FUNCTION_BLOCK "TYPIC_C106_IF_TFO"   // FB80, FBD
TITLE = TYPIC_C106_IF_TFO: Transformator
{ S7_Optimized_Access := 'TRUE' }
AUTHOR : OCOTECH
FAMILY : Typical
NAME : C106.704
// Logisch Object Besturing: C106.704
// 
// De interne functie Transformator verzorgt de bewaking van een transformator.
// stored: MemoryReserve 10, SetENOAutomatically false
   VAR_INPUT
      EXT_AUT { ExternalAccessible := 'False'; ExternalVisible := 'False'; ExternalWritable := 'False'} : Bool;   // Externe (hoofd) beveiliging (1 = OK)
      EXT_HW { ExternalAccessible := 'False'; ExternalVisible := 'False'; ExternalWritable := 'False'} : Bool;   // Sturings hardware (PLC) bewaking (1 = OK)
      IN_STO_NOK { ExternalAccessible := 'False'; ExternalVisible := 'False'; ExternalWritable := 'False'} : Bool;   // Storing aanwezig die niet observeerbaar tot gevolg heeft
      IN_STO_OK { ExternalAccessible := 'False'; ExternalVisible := 'False'; ExternalWritable := 'False'} : Bool;   // Storing aanwezig die observeerbaarheid niet beinvloed
      IN_TFO_BSC1 { ExternalAccessible := 'False'; ExternalVisible := 'False'; ExternalWritable := 'False'} : Bool;   // Transformator beschikbaar
      IN_TFO_BSC2 { ExternalAccessible := 'False'; ExternalVisible := 'False'; ExternalWritable := 'False'} : Bool;   // Transformator niet beschikbaar
      IN_TFO_BSC3 { ExternalAccessible := 'False'; ExternalVisible := 'False'; ExternalWritable := 'False'} : Bool;   // Transformator beperkt beschikbaar
      IN_AUT_C106 { ExternalAccessible := 'False'; ExternalVisible := 'False'; ExternalWritable := 'False'} : Bool;   // Beveiligingen: serie geschakelde terugmelding (1 = OK)
   END_VAR
   VAR_OUTPUT
      VAR_IF_NME { ExternalAccessible := 'False'; ExternalVisible := 'False'; ExternalWritable := 'False'} : "C106_VAR_IF_NME_TYPIC";   // Struct met alle variabelen naar bovenliggende functies
   END_VAR
   VAR
      STO { ExternalWritable := 'False'} : Struct   // Storingen
         A001 : Bool;   // Beveiliging aangesproken
         A002 : Bool;   // Hoogspanningstransformator in storing
         A003 : Bool;   // Algemene storing hoogspanningstransformator
      END_STRUCT;
      VAR { ExternalWritable := 'False'} : Struct   // Variabelen
         BSC1 { ExternalAccessible := 'False'; ExternalVisible := 'False'} : Bool;   // Transformator beschikbaar
         BSC2 { ExternalAccessible := 'False'; ExternalVisible := 'False'} : Bool;   // Transformator niet beschikbaar
         BSC3 { ExternalAccessible := 'False'; ExternalVisible := 'False'} : Bool;   // Transformator beperkt beschikbaar
         EXT_AUT { ExternalAccessible := 'False'; ExternalVisible := 'False'} : Bool;   // Externe (hoofd) beveiliging aangesproken
         EXT_HW { ExternalAccessible := 'False'; ExternalVisible := 'False'} : Bool;   // Sturings hardware (PLC) in storing
      END_STRUCT;
   END_VAR
BEGIN

REGION Network 1: START
END_REGION

REGION Network 2: +++ Verwerking meetwaarden en statussen +++
   // De meetwaarde en status wordt ontvangen vanuit de interne sturing.
END_REGION

REGION Network 3: +++ Storingen +++
   // Verwerken van de storingsmeldingen (inputs).
END_REGION

REGION Network 4: Storing A001: Beveiliging aangesproken
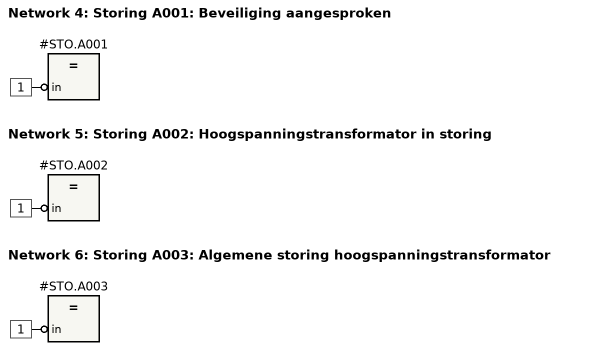
   #STO.A001 := NOT 1;
END_REGION

REGION Network 5: Storing A002: Hoogspanningstransformator in storing
   #STO.A002 := NOT 1;
END_REGION

REGION Network 6: Storing A003: Algemene storing hoogspanningstransformator
   #STO.A003 := NOT 1;
END_REGION

REGION Network 7 (SCL): EINDE
   // Variabelen van intern scada rakvlak naar outputs copieren
   #VAR_IF_NME.BSC1 := #VAR.BSC1;
   #VAR_IF_NME.BSC2 := #VAR.BSC2;
   #VAR_IF_NME.BSC3 := #VAR.BSC3;
   #VAR_IF_NME.EXT_AUT := #VAR.EXT_AUT;
   #VAR_IF_NME.EXT_HW := #VAR.EXT_HW;
END_REGION
END_FUNCTION_BLOCK

FUNCTION_BLOCK "TYPIC_C103_BF_LSK"   // FB21, FBD
TITLE = TYPIC_C103_BF_LSK: Laagspanning koker
{ S7_Optimized_Access := 'TRUE' }
AUTHOR : OCOTECH
FAMILY : Typical
NAME : C103.801
// Logisch Object Besturing: C103.801
// 
// Het doel van de BF LSK (laagspanning koker) is om de algemene opvolging te voorzien van de laagspanningsinstallatie per verkeerskoker.
// stored: MemoryReserve 10, SetENOAutomatically false
   VAR_INPUT
      STU_ALG_LCK_SIG { ExternalAccessible := 'False'; ExternalVisible := 'False'; ExternalWritable := 'False'} : USInt;   // Onderdruk alarmen
   END_VAR
   VAR_IN_OUT
      VAR_REL : Array[0..1] of Bool;   // Array met de standmeldingen van alle vermogenschakelaars
   END_VAR
   VAR
      SIG { ExternalWritable := 'False'} : Struct   // Signaleringen
         AA01 : Bool;   // Laagspanningsinstallatie niet observeerbaar
         AA02 : Bool;   // Laagspanningsinstallatie storing algemeen
         A001 : Bool;   // Laagspanningsinstallatie standmelding beveiliging uit
         AB01 : Bool;   // Laagspanningsinstallatie niet beschikbaar
         AB02 : Bool;   // Laagspanningsinstallatie beperkt beschikbaar
      END_STRUCT;
      VAR { ExternalWritable := 'False'} : Struct   // Variabelen
         BSC : USInt;   // Geeft de beschikbaarheid aan van het deelsysteem
         LSK_STS : USInt;   // De status van het deelsysteem
         VGV_SIG_VOP : Bool;   // TRUE = Signaleringen vrijgegeven voor verkeersoperator FALSE = Onderdrukt
      END_STRUCT;
   END_VAR
BEGIN

REGION Network 1: START
END_REGION

REGION Network 2: +++ Bepalen beschikbaarheidsstatus +++
   // Beschikbaarheidsstatus (beschikbaar / beperkt beschikbaar / niet beschikbaar) bepalen.
END_REGION

REGION Network 3 (SCL): Beschikbaarheidsstatus bepalen
   IF 
       //voorwaarden "Niet beschikbaar"
       TRUE
   THEN
       //Beschikbaarheidsstatus = Niet Beschikbaar
       #VAR.BSC:= "NietBeschikbaar";
   ELSIF
       //voorwaarden "Beperkt beschikbaar"
       TRUE
   THEN
       //Beschikbaarheidsstatus = Beperkt Beschikbaar
       #VAR.BSC:= "Beperkt";
   ELSE
       //Beschikbaarheidsstatus = Beschikbaar
       #VAR.BSC:= "Beschikbaar";
   END_IF;
END_REGION

REGION Network 4: +++ Signaleringen +++
   // Aanmaken signaleringen
END_REGION

REGION Network 5: Signalering AB01 : Niet Beschikbaar
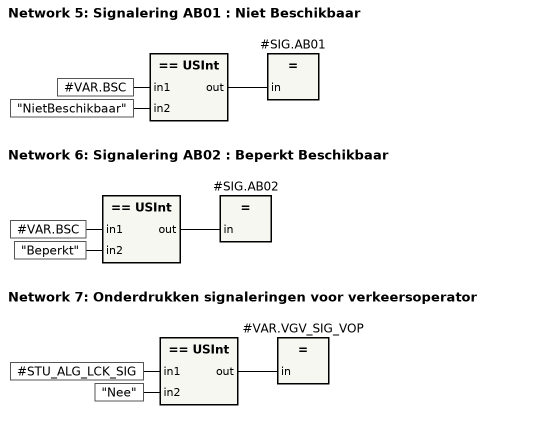
   #SIG.AB01 := #VAR.BSC = "NietBeschikbaar";
END_REGION

REGION Network 6: Signalering AB02 : Beperkt Beschikbaar
   #SIG.AB02 := #VAR.BSC = "Beperkt";
END_REGION

REGION Network 7: Onderdrukken signaleringen voor verkeersoperator
   // Via de variabele VGV_SIG_VOP wordt aan IRIS SCADA doorgegeven of signaleringen (bestemd voor de verkeersoperator) van de deze functie zichtbaar (of onderdrukt) moeten zijn.
   #VAR.VGV_SIG_VOP := #STU_ALG_LCK_SIG = "Nee";
END_REGION

REGION Network 8: +++ Doorkoppeling energieverbruik en vermogen LSK +++
   // De actuele vermogen en energiemeting wordt doorgegeven aan de coordinerende functie Energievoorziening.
END_REGION

REGION Network 9: EINDE
   // Variabelen van intern scada rakvlak naar outputs copieren
END_REGION
END_FUNCTION_BLOCK

FUNCTION_BLOCK "TYPIC_C103_IF_HVI"   // FB20, FBD
TITLE = TYPIC_C103_IF_HVI: ALSB
{ S7_Optimized_Access := 'TRUE' }
AUTHOR : OCOTECH
FAMILY : Typical
NAME : C103.701
// Logisch Object Besturing: C103.802
// 
// De interne functie laagspanningsverdeelbord verzorgt de bewaking van een laagspanningsverdeelbord.
// stored: MemoryReserve 10, SetENOAutomatically false
   VAR_INPUT
      EXT_AUT { ExternalAccessible := 'False'; ExternalVisible := 'False'; ExternalWritable := 'False'} : Bool;   // Externe (hoofd) beveiliging (1 = OK)
      EXT_HW { ExternalAccessible := 'False'; ExternalVisible := 'False'; ExternalWritable := 'False'} : Bool;   // Sturings hardware (PLC) bewaking (1 = OK)
      IN_PWR1 { ExternalAccessible := 'False'; ExternalVisible := 'False'; ExternalWritable := 'False'} : Real;   // Actief vermogen
      IN_PWR2 { ExternalAccessible := 'False'; ExternalVisible := 'False'; ExternalWritable := 'False'} : Real;   // Reactief vermogen
      IN_SPA_1 { ExternalAccessible := 'False'; ExternalVisible := 'False'; ExternalWritable := 'False'} : Real;   // Spanningsniveau lijn 1
      IN_SPA_2 { ExternalAccessible := 'False'; ExternalVisible := 'False'; ExternalWritable := 'False'} : Real;   // Spanningsniveau lijn 2
      IN_SPA_3 { ExternalAccessible := 'False'; ExternalVisible := 'False'; ExternalWritable := 'False'} : Real;   // Spanningsniveau lijn 3
      IN_SPA_4 { ExternalAccessible := 'False'; ExternalVisible := 'False'; ExternalWritable := 'False'} : Real;   // Lijnspanning L1-L2
      IN_SPA_5 { ExternalAccessible := 'False'; ExternalVisible := 'False'; ExternalWritable := 'False'} : Real;   // Lijnspanning L2-L3
      IN_SPA_6 { ExternalAccessible := 'False'; ExternalVisible := 'False'; ExternalWritable := 'False'} : Real;   // Lijnspanning L1-L3
      IN_STR_1 { ExternalAccessible := 'False'; ExternalVisible := 'False'; ExternalWritable := 'False'} : Real;   // Stroom lijn 1
      IN_STR_2 { ExternalAccessible := 'False'; ExternalVisible := 'False'; ExternalWritable := 'False'} : Real;   // Stroom lijn 2
      IN_STR_3 { ExternalAccessible := 'False'; ExternalVisible := 'False'; ExternalWritable := 'False'} : Real;   // Stroom lijn 3
      IN_STR_4 { ExternalAccessible := 'False'; ExternalVisible := 'False'; ExternalWritable := 'False'} : Real;   // Stroom nulleider
      IN_PHI { ExternalAccessible := 'False'; ExternalVisible := 'False'; ExternalWritable := 'False'} : Real;   // Arbeidsfactor
      IN_BEV_SPA { ExternalAccessible := 'False'; ExternalVisible := 'False'; ExternalWritable := 'False'} : Bool;   // Status beveiliging detectie railspanning
      IN_SPA2 { ExternalAccessible := 'False'; ExternalVisible := 'False'; ExternalWritable := 'False'} : Bool;   // Status detectie railspanning
      IN_SPA1_STO { ExternalAccessible := 'False'; ExternalVisible := 'False'; ExternalWritable := 'False'} : Bool;   // Status detectie railspanning
      IN_PHI_OK { ExternalAccessible := 'False'; ExternalVisible := 'False'; ExternalWritable := 'False'} : Bool;   // Status fasebewaking
      IN_HLP_OK { ExternalAccessible := 'False'; ExternalVisible := 'False'; ExternalWritable := 'False'} : Bool;   // Status hulpvoedingen (groepscontact)
      IN_SPD_OK { ExternalAccessible := 'False'; ExternalVisible := 'False'; ExternalWritable := 'False'} : Bool;   // Status overspanningsbeveiliging
      IN_SPA3_STO { ExternalAccessible := 'False'; ExternalVisible := 'False'; ExternalWritable := 'False'} : Bool;   // Status storing detectie railspanning
      IN_SPA4_STO { ExternalAccessible := 'False'; ExternalVisible := 'False'; ExternalWritable := 'False'} : Bool;   // Status storing detectie railspanning
      IN_STS1 { ExternalAccessible := 'False'; ExternalVisible := 'False'; ExternalWritable := 'False'} : Bool;   // Status van elke schuif [IN]
      IN_STS2 { ExternalAccessible := 'False'; ExternalVisible := 'False'; ExternalWritable := 'False'} : Bool;   // Status van elke schuif [TEST]
      IN_STS3 { ExternalAccessible := 'False'; ExternalVisible := 'False'; ExternalWritable := 'False'} : Bool;   // Status van elke schuif [UIT]
      IN_AUT_TOE { ExternalAccessible := 'False'; ExternalVisible := 'False'; ExternalWritable := 'False'} : Bool;   // Standmelding van elke vermogenschakelaar TOE [gesloten]
      IN_OK { ExternalAccessible := 'False'; ExternalVisible := 'False'; ExternalWritable := 'False'} : Bool;   // Standmelding beveiliging vertrek
   END_VAR
   VAR_OUTPUT
      VAR_IF_HVI { ExternalAccessible := 'False'; ExternalVisible := 'False'; ExternalWritable := 'False'} : "C103_VAR_IF_HVI_TYPIC";   // Struct met alle variabelen naar bovenliggende functies
   END_VAR
   VAR
      STO { ExternalWritable := 'False'} : Struct   // Storingen
         A001 { ExternalAccessible := 'False'; ExternalVisible := 'False'} : Bool;   // Laagspanningsverdeelbord beveiliging aangesproken
         A002 { ExternalAccessible := 'False'; ExternalVisible := 'False'} : Bool;   // Laagspanningsverdeelbord in storing
      END_STRUCT;
      VAR { ExternalWritable := 'False'} : Struct   // Variabelen
         PWR1 { ExternalAccessible := 'False'; ExternalVisible := 'False'} : Real;   // Actief vermogen
         PWR2 { ExternalAccessible := 'False'; ExternalVisible := 'False'} : Real;   // Reactief vermogen
         SPA_1 { ExternalAccessible := 'False'; ExternalVisible := 'False'} : Real;   // Spanningsniveau lijn 1
         SPA_2 { ExternalAccessible := 'False'; ExternalVisible := 'False'} : Real;   // Spanningsniveau lijn 2
         SPA_3 { ExternalAccessible := 'False'; ExternalVisible := 'False'} : Real;   // Spanningsniveau lijn 3
         SPA_4 { ExternalAccessible := 'False'; ExternalVisible := 'False'} : Real;   // Lijnspanning L1-L2
         SPA_5 { ExternalAccessible := 'False'; ExternalVisible := 'False'} : Real;   // Lijnspanning L2-L3
         SPA_6 { ExternalAccessible := 'False'; ExternalVisible := 'False'} : Real;   // Lijnspanning L1-L3
         STR_1 { ExternalAccessible := 'False'; ExternalVisible := 'False'} : Real;   // Stroom lijn 1
         STR_2 { ExternalAccessible := 'False'; ExternalVisible := 'False'} : Real;   // Stroom lijn 2
         STR_3 { ExternalAccessible := 'False'; ExternalVisible := 'False'} : Real;   // Stroom lijn 3
         STR_4 { ExternalAccessible := 'False'; ExternalVisible := 'False'} : Real;   // Stroom nulleider
         PHI { ExternalAccessible := 'False'; ExternalVisible := 'False'} : Real;   // Arbeidsfactor
         BEV_SPA { ExternalAccessible := 'False'; ExternalVisible := 'False'} : Bool;   // Status beveiliging detectie railspanning
         SPA2 { ExternalAccessible := 'False'; ExternalVisible := 'False'} : Bool;   // Status detectie railspanning
         SPA1_STO { ExternalAccessible := 'False'; ExternalVisible := 'False'} : Bool;   // Status detectie railspanning
         PHI_OK { ExternalAccessible := 'False'; ExternalVisible := 'False'} : Bool;   // Status fasebewaking
         HLP_OK { ExternalAccessible := 'False'; ExternalVisible := 'False'} : Bool;   // Status hulpvoedingen (groepscontact)
         SPD_OK { ExternalAccessible := 'False'; ExternalVisible := 'False'} : Bool;   // Status overspanningsbeveiliging
         SPA3_STO { ExternalAccessible := 'False'; ExternalVisible := 'False'} : Bool;   // Status storing detectie railspanning
         SPA4_STO { ExternalAccessible := 'False'; ExternalVisible := 'False'} : Bool;   // Status storing detectie railspanning
         STS1 { ExternalAccessible := 'False'; ExternalVisible := 'False'} : Bool;   // Status van elke schuif [IN]
         STS2 { ExternalAccessible := 'False'; ExternalVisible := 'False'} : Bool;   // Status van elke schuif [TEST]
         STS3 { ExternalAccessible := 'False'; ExternalVisible := 'False'} : Bool;   // Status van elke schuif [UIT]
         AUT_TOE { ExternalAccessible := 'False'; ExternalVisible := 'False'} : Bool;   // Standmelding van elke vermogenschakelaar TOE [gesloten]
         BEV_OK : Bool;
      END_STRUCT;
   END_VAR
BEGIN

REGION Network 1: START
END_REGION

REGION Network 2: +++ Verwerking meetwaarden en statussen +++
   // De meetwaarde en status wordt ontvangen vanuit de interne sturing.
END_REGION

REGION Network 3: +++ Storingen +++
   // Combinatie van de storingen
END_REGION

REGION Network 4: Storing A001: Laagspanningsverdeelbord beveiliging aangesproken
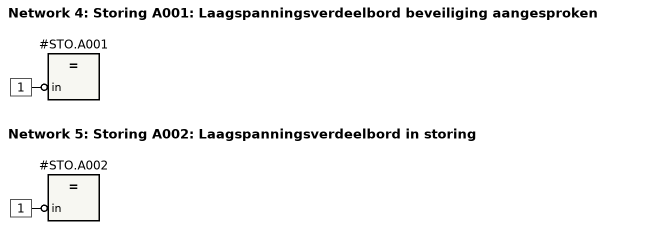
   #STO.A001 := NOT 1;
END_REGION

REGION Network 5: Storing A002: Laagspanningsverdeelbord in storing
   #STO.A002 := NOT 1;
END_REGION

REGION Network 6 (SCL): EINDE
   // Variabelen van intern scada rakvlak naar outputs copieren
   #VAR_IF_HVI.PWR1 := #VAR.PWR1;
   #VAR_IF_HVI.PWR2 := #VAR.PWR2;
   #VAR_IF_HVI.SPA_1 := #VAR.SPA_1;
   #VAR_IF_HVI.SPA_2 := #VAR.SPA_2;
   #VAR_IF_HVI.SPA_3 := #VAR.SPA_3;
   #VAR_IF_HVI.SPA_4 := #VAR.SPA_4;
   #VAR_IF_HVI.SPA_5 := #VAR.SPA_5;
   #VAR_IF_HVI.SPA_6 := #VAR.SPA_6;
   #VAR_IF_HVI.STR_1 := #VAR.STR_1;
   #VAR_IF_HVI.STR_2 := #VAR.STR_2;
   #VAR_IF_HVI.STR_3 := #VAR.STR_3;
   #VAR_IF_HVI.STR_4 := #VAR.STR_4;
   #VAR_IF_HVI.PHI := #VAR.PHI;
   #VAR_IF_HVI.BEV_SPA := #VAR.BEV_SPA;
   #VAR_IF_HVI.SPA2 := #VAR.SPA2;
   #VAR_IF_HVI.SPA1_STO := #VAR.SPA1_STO;
   #VAR_IF_HVI.PHI_OK := #VAR.PHI_OK;
   #VAR_IF_HVI.HLP_OK := #VAR.HLP_OK;
   #VAR_IF_HVI.SPD_OK := #VAR.SPD_OK;
   #VAR_IF_HVI.SPA3_STO := #VAR.SPA3_STO;
   #VAR_IF_HVI.SPA4_STO := #VAR.SPA4_STO;
   #VAR_IF_HVI.STS1 := #VAR.STS1;
   #VAR_IF_HVI.STS2 := #VAR.STS2;
   #VAR_IF_HVI.STS3 := #VAR.STS3;
   #VAR_IF_HVI.AUT_TOE := #VAR.AUT_TOE;
   #VAR_IF_HVI.BEV_OK := #VAR.BEV_OK;
END_REGION
END_FUNCTION_BLOCK

FUNCTION_BLOCK "TYPIC_C103_IF_HVN"   // FB18, FBD
TITLE = TYPIC_C103_IF_HVN: ALSB NB
{ S7_Optimized_Access := 'TRUE' }
AUTHOR : OCOTECH
FAMILY : Typical
NAME : C103.702
// Logisch Object Besturing: C103.803
// 
// De interne functie laagspanningsverdeelbord no break verzorgt de bewaking van een laagspanningsverdeelbord no break.
// stored: MemoryReserve 10, SetENOAutomatically false
   VAR_INPUT
      EXT_AUT { ExternalAccessible := 'False'; ExternalVisible := 'False'; ExternalWritable := 'False'} : Bool;   // Externe (hoofd) beveiliging (1 = OK)
      EXT_HW { ExternalAccessible := 'False'; ExternalVisible := 'False'; ExternalWritable := 'False'} : Bool;   // Sturings hardware (PLC) bewaking (1 = OK)
      IN_PWR1 { ExternalAccessible := 'False'; ExternalVisible := 'False'; ExternalWritable := 'False'} : Real;   // Actief vermogen
      IN_PWR2 { ExternalAccessible := 'False'; ExternalVisible := 'False'; ExternalWritable := 'False'} : Real;   // Reactief vermogen
      IN_SPA_1 { ExternalAccessible := 'False'; ExternalVisible := 'False'; ExternalWritable := 'False'} : Real;   // Spanningsniveau lijn 1
      IN_SPA_2 { ExternalAccessible := 'False'; ExternalVisible := 'False'; ExternalWritable := 'False'} : Real;   // Spanningsniveau lijn 2
      IN_SPA_3 { ExternalAccessible := 'False'; ExternalVisible := 'False'; ExternalWritable := 'False'} : Real;   // Spanningsniveau lijn 3
      IN_SPA_4 { ExternalAccessible := 'False'; ExternalVisible := 'False'; ExternalWritable := 'False'} : Real;   // Lijnspanning L1-L2
      IN_SPA_5 { ExternalAccessible := 'False'; ExternalVisible := 'False'; ExternalWritable := 'False'} : Real;   // Lijnspanning L2-L3
      IN_SPA_6 { ExternalAccessible := 'False'; ExternalVisible := 'False'; ExternalWritable := 'False'} : Real;   // Lijnspanning L1-L3
      IN_STR_1 { ExternalAccessible := 'False'; ExternalVisible := 'False'; ExternalWritable := 'False'} : Real;   // Stroom lijn 1
      IN_STR_2 { ExternalAccessible := 'False'; ExternalVisible := 'False'; ExternalWritable := 'False'} : Real;   // Stroom lijn 2
      IN_STR_3 { ExternalAccessible := 'False'; ExternalVisible := 'False'; ExternalWritable := 'False'} : Real;   // Stroom lijn 3
      IN_STR_4 { ExternalAccessible := 'False'; ExternalVisible := 'False'; ExternalWritable := 'False'} : Real;   // Stroom nulleider
      IN_PHI { ExternalAccessible := 'False'; ExternalVisible := 'False'; ExternalWritable := 'False'} : Real;   // Arbeidsfactor
      IN_AUT_TOE { ExternalAccessible := 'False'; ExternalVisible := 'False'; ExternalWritable := 'False'} : Bool;   // Standmelding van elke vermogenschakelaar TOE [gesloten]
      IN_SCL1 { ExternalAccessible := 'False'; ExternalVisible := 'False'; ExternalWritable := 'False'} : Bool;   // Standmelding externe bypass netspanning
      IN_SCL2 { ExternalAccessible := 'False'; ExternalVisible := 'False'; ExternalWritable := 'False'} : Bool;   // Standmelding aankomstschakelaar UPS
   END_VAR
   VAR_OUTPUT
      VAR_IF_HVN { ExternalAccessible := 'False'; ExternalVisible := 'False'; ExternalWritable := 'False'} : "C103_VAR_IF_HVN_TYPIC";   // Struct met alle variabelen naar bovenliggende functies
   END_VAR
   VAR
      STO { ExternalWritable := 'False'} : Struct   // Storingen
         A001 { ExternalAccessible := 'False'; ExternalVisible := 'False'} : Bool;   // Laagspanningsverdeelbord no break beveiliging aangesproken
         A002 { ExternalAccessible := 'False'; ExternalVisible := 'False'} : Bool;   // Laagspanningsverdeelbord no break in storing
      END_STRUCT;
      VAR { ExternalWritable := 'False'} : Struct   // Variabelen
         PWR1 { ExternalAccessible := 'False'; ExternalVisible := 'False'} : Real;   // Actief vermogen
         PWR2 { ExternalAccessible := 'False'; ExternalVisible := 'False'} : Real;   // Reactief vermogen
         SPA_1 { ExternalAccessible := 'False'; ExternalVisible := 'False'} : Real;   // Spanningsniveau lijn 1
         SPA_2 { ExternalAccessible := 'False'; ExternalVisible := 'False'} : Real;   // Spanningsniveau lijn 2
         SPA_3 { ExternalAccessible := 'False'; ExternalVisible := 'False'} : Real;   // Spanningsniveau lijn 3
         SPA_4 { ExternalAccessible := 'False'; ExternalVisible := 'False'} : Real;   // Lijnspanning L1-L2
         SPA_5 { ExternalAccessible := 'False'; ExternalVisible := 'False'} : Real;   // Lijnspanning L2-L3
         SPA_6 { ExternalAccessible := 'False'; ExternalVisible := 'False'} : Real;   // Lijnspanning L1-L3
         STR_1 { ExternalAccessible := 'False'; ExternalVisible := 'False'} : Real;   // Stroom lijn 1
         STR_2 { ExternalAccessible := 'False'; ExternalVisible := 'False'} : Real;   // Stroom lijn 2
         STR_3 { ExternalAccessible := 'False'; ExternalVisible := 'False'} : Real;   // Stroom lijn 3
         STR_4 { ExternalAccessible := 'False'; ExternalVisible := 'False'} : Real;   // Stroom nulleider
         PHI { ExternalAccessible := 'False'; ExternalVisible := 'False'} : Real;   // Arbeidsfactor
         AUT_TOE { ExternalAccessible := 'False'; ExternalVisible := 'False'} : Bool;   // Standmelding van elke vermogenschakelaar TOE [gesloten]
         SCL1 { ExternalAccessible := 'False'; ExternalVisible := 'False'} : Bool;   // Standmelding externe bypass netspanning
         SCL2 { ExternalAccessible := 'False'; ExternalVisible := 'False'} : Bool;   // Standmelding aankomstschakelaar UPS
      END_STRUCT;
   END_VAR
BEGIN

REGION Network 1: START
END_REGION

REGION Network 2: +++ Verwerking meetwaarden en statussen +++
   // De meetwaarde en status wordt ontvangen vanuit de interne sturing.
END_REGION

REGION Network 3: +++ Storingen +++
   // Combinatie van de storingen
END_REGION

REGION Network 4: Storing A001: Laagspanningsverdeelbord no break beveiliging aangesproken
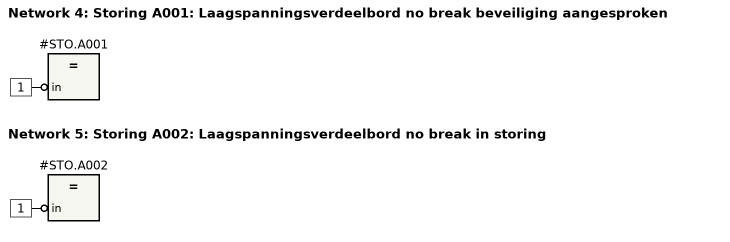
   #STO.A001 := NOT 1;
END_REGION

REGION Network 5: Storing A002: Laagspanningsverdeelbord no break in storing
   #STO.A002 := NOT 1;
END_REGION

REGION Network 6 (SCL): EINDE
   // Variabelen van intern scada rakvlak naar outputs copieren
   #VAR_IF_HVN.PWR1 := #VAR.PWR1;
   #VAR_IF_HVN.PWR2 := #VAR.PWR2;
   #VAR_IF_HVN.SPA_1 := #VAR.SPA_1;
   #VAR_IF_HVN.SPA_2 := #VAR.SPA_2;
   #VAR_IF_HVN.SPA_3 := #VAR.SPA_3;
   #VAR_IF_HVN.SPA_4 := #VAR.SPA_4;
   #VAR_IF_HVN.SPA_5 := #VAR.SPA_5;
   #VAR_IF_HVN.SPA_6 := #VAR.SPA_6;
   #VAR_IF_HVN.STR_1 := #VAR.STR_1;
   #VAR_IF_HVN.STR_2 := #VAR.STR_2;
   #VAR_IF_HVN.STR_3 := #VAR.STR_3;
   #VAR_IF_HVN.STR_4 := #VAR.STR_4;
   #VAR_IF_HVN.PHI := #VAR.PHI;
   #VAR_IF_HVN.AUT_TOE := #VAR.AUT_TOE;
   #VAR_IF_HVN.SCL1 := #VAR.SCL1;
   #VAR_IF_HVN.SCL2 := #VAR.SCL2;
END_REGION
END_FUNCTION_BLOCK

FUNCTION_BLOCK "TYPIC_C103_IF_OVB"   // FB32, FBD
TITLE = TYPIC_C103_IF_OVB: LSBB
{ S7_Optimized_Access := 'TRUE' }
AUTHOR : OCOTECH
FAMILY : Typical
NAME : C103.705
// Logisch Object Besturing: C103.805
// 
// De interne functie laagspanningsverdeelbord buiten verzorgt de bewaking van een laagspanningsverdeelbord buiten.
// stored: MemoryReserve 10, SetENOAutomatically false
   VAR_INPUT
      EXT_AUT { ExternalAccessible := 'False'; ExternalVisible := 'False'; ExternalWritable := 'False'} : Bool;   // Externe (hoofd) beveiliging (1 = OK)
      EXT_HW { ExternalAccessible := 'False'; ExternalVisible := 'False'; ExternalWritable := 'False'} : Bool;   // Sturings hardware (PLC) bewaking (1 = OK)
      IN_SCL { ExternalAccessible := 'False'; ExternalVisible := 'False'; ExternalWritable := 'False'} : Bool;   // LSB ingangszone 400V/230V
   END_VAR
   VAR_OUTPUT
      VAR_IF_OVB { ExternalAccessible := 'False'; ExternalVisible := 'False'; ExternalWritable := 'False'} : "C103_VAR_IF_OVB_TYPIC";   // Struct met alle variabelen naar bovenliggende functies
   END_VAR
   VAR
      STO { ExternalWritable := 'False'} : Struct   // Storingen
         A001 { ExternalAccessible := 'False'; ExternalVisible := 'False'} : Bool;   // Laagspanningsverdeelbord buiten beveiliging aangesproken
         A002 { ExternalAccessible := 'False'; ExternalVisible := 'False'} : Bool;   // Laagspanningsverdeelbord buiten in dienstkoker in storing
      END_STRUCT;
      VAR { ExternalWritable := 'False'} : Struct   // Variabelen
         SCL { ExternalAccessible := 'False'; ExternalVisible := 'False'} : Bool;   // Standmelding ingangszone 400V/230V
      END_STRUCT;
   END_VAR
BEGIN

REGION Network 1: START
END_REGION

REGION Network 2: +++ Verwerking meetwaarden en statussen +++
   // De meetwaarde en status wordt ontvangen vanuit de interne sturing.
END_REGION

REGION Network 3: +++ Storingen +++
   // Combinatie van de storingen
END_REGION

REGION Network 4: Storing A001: Laagspanningsverdeelbord buiten beveiliging aangesproken
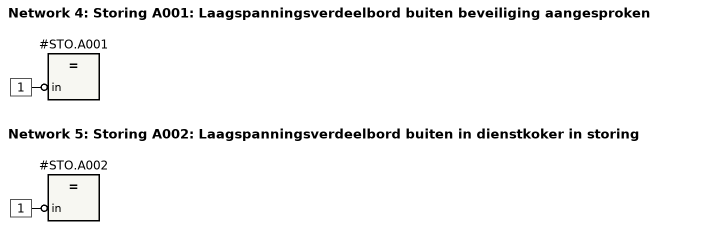
   #STO.A001 := NOT 1;
END_REGION

REGION Network 5: Storing A002: Laagspanningsverdeelbord buiten in dienstkoker in storing
   #STO.A002 := NOT 1;
END_REGION

REGION Network 6 (SCL): EINDE
   // Variabelen van intern scada rakvlak naar outputs copieren
   #VAR_IF_OVB.SCL := #VAR.SCL;
END_REGION
END_FUNCTION_BLOCK

FUNCTION_BLOCK "TYPIC_C103_IF_OVI"   // FB17, FBD
TITLE = TYPIC_C103_IF_OVI: LSB
{ S7_Optimized_Access := 'TRUE' }
AUTHOR : OCOTECH
FAMILY : Typical
NAME : C103.703
// Logisch Object Besturing: C103.802
// 
// De interne functie laagspanningsverdeelbord in dienstkoker verzorgt de bewaking van een laagspanningsverdeelbord in dienstkoker.
// stored: MemoryReserve 10, SetENOAutomatically false
   VAR_INPUT
      EXT_AUT { ExternalAccessible := 'False'; ExternalVisible := 'False'; ExternalWritable := 'False'} : Bool;   // Externe (hoofd) beveiliging (1 = OK)
      EXT_HW { ExternalAccessible := 'False'; ExternalVisible := 'False'; ExternalWritable := 'False'} : Bool;   // Sturings hardware (PLC) bewaking (1 = OK)
      IN_SCL { ExternalAccessible := 'False'; ExternalVisible := 'False'; ExternalWritable := 'False'} : Bool;   // Standmelding aankomstschakelaar
   END_VAR
   VAR_OUTPUT
      VAR_IF_OVI { ExternalAccessible := 'False'; ExternalVisible := 'False'; ExternalWritable := 'False'} : "C103_VAR_IF_OVI_TYPIC";   // Struct met alle variabelen naar bovenliggende functies
   END_VAR
   VAR
      STO { ExternalWritable := 'False'} : Struct   // Storingen
         A001 { ExternalAccessible := 'False'; ExternalVisible := 'False'} : Bool;   // Laagspanningsverdeelbord beveiliging aangesproken
         A002 { ExternalAccessible := 'False'; ExternalVisible := 'False'} : Bool;   // Laagspanningsverdeelbord in storing
      END_STRUCT;
      VAR { ExternalWritable := 'False'} : Struct   // Variabelen
         SCL { ExternalAccessible := 'False'; ExternalVisible := 'False'} : Bool;   // Standmelding aankomstschakelaar
      END_STRUCT;
   END_VAR
BEGIN

REGION Network 1: START
END_REGION

REGION Network 2: +++ Verwerking meetwaarden en statussen +++
   // De meetwaarde en status wordt ontvangen vanuit de interne sturing.
END_REGION

REGION Network 3: +++ Storingen +++
   // Combinatie van de storingen
END_REGION

REGION Network 4: Storing A001: Laagspanningsverdeelbord beveiliging aangesproken
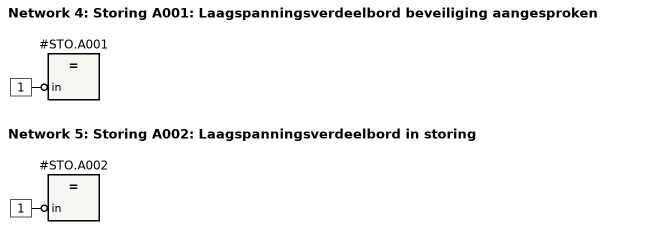
   #STO.A001 := NOT 1;
END_REGION

REGION Network 5: Storing A002: Laagspanningsverdeelbord in storing
   #STO.A002 := NOT 1;
END_REGION

REGION Network 6 (SCL): EINDE
   // Variabelen van intern scada rakvlak naar outputs copieren
   #VAR_IF_OVI.SCL := #VAR.SCL;
END_REGION
END_FUNCTION_BLOCK

FUNCTION_BLOCK "TYPIC_C103_IF_OVN"   // FB16, FBD
TITLE = TYPIC_C103_IF_OVN: LSB NB
{ S7_Optimized_Access := 'TRUE' }
AUTHOR : OCOTECH
FAMILY : Typical
NAME : C103.704
// Logisch Object Besturing: C103.805
// 
// De interne functie laagspanningsverdeelbord no break in dienstkoker verzorgt de bewaking van een laagspanningsverdeelbord no break in dienstkoker.
// stored: MemoryReserve 10, SetENOAutomatically false
   VAR_INPUT
      EXT_AUT { ExternalAccessible := 'False'; ExternalVisible := 'False'; ExternalWritable := 'False'} : Bool;   // Externe (hoofd) beveiliging (1 = OK)
      EXT_HW { ExternalAccessible := 'False'; ExternalVisible := 'False'; ExternalWritable := 'False'} : Bool;   // Sturings hardware (PLC) bewaking (1 = OK)
      IN_SCL1 { ExternalAccessible := 'False'; ExternalVisible := 'False'; ExternalWritable := 'False'} : Bool;   // Standmelding aankomstschakelaar normaal
      IN_SCL2 { ExternalAccessible := 'False'; ExternalVisible := 'False'; ExternalWritable := 'False'} : Bool;   // Standmelding aankomstschakelaar no-break
      IN_BEV { ExternalAccessible := 'False'; ExternalVisible := 'False'; ExternalWritable := 'False'} : Bool;   // Standmelding automaat kast verwarming en ventilatie
   END_VAR
   VAR_OUTPUT
      VAR_IF_OVN { ExternalAccessible := 'False'; ExternalVisible := 'False'; ExternalWritable := 'False'} : "C103_VAR_IF_OVN_TYPIC";   // Struct met alle variabelen naar bovenliggende functies
   END_VAR
   VAR
      STO { ExternalWritable := 'False'} : Struct   // Storingen
         A001 { ExternalAccessible := 'False'; ExternalVisible := 'False'} : Bool;   // Laagspanningsverdeelbord no break in dienstkoker beveiliging aangesproken
         A002 { ExternalAccessible := 'False'; ExternalVisible := 'False'} : Bool;   // Laagspanningsverdeelbord no break in dienstkoker in storing
      END_STRUCT;
      VAR { ExternalWritable := 'False'} : Struct   // Variabelen
         SCL1 { ExternalAccessible := 'False'; ExternalVisible := 'False'} : Bool;   // Standmelding aankomstschakelaar normaal
         SCL2 { ExternalAccessible := 'False'; ExternalVisible := 'False'} : Bool;   // Standmelding aankomstschakelaar no-break
         BEV { ExternalAccessible := 'False'; ExternalVisible := 'False'} : Bool;   // Standmelding automaat kast verwarming en ventilatie
      END_STRUCT;
   END_VAR
BEGIN

REGION Network 1: START
END_REGION

REGION Network 2: +++ Verwerking meetwaarden en statussen +++
   // De meetwaarde en status wordt ontvangen vanuit de interne sturing.
END_REGION

REGION Network 3: +++ Storingen +++
   // Combinatie van de storingen
END_REGION

REGION Network 4: Storing A001: Laagspanningsverdeelbord no break in dienstkoker beveiliging aangesproken
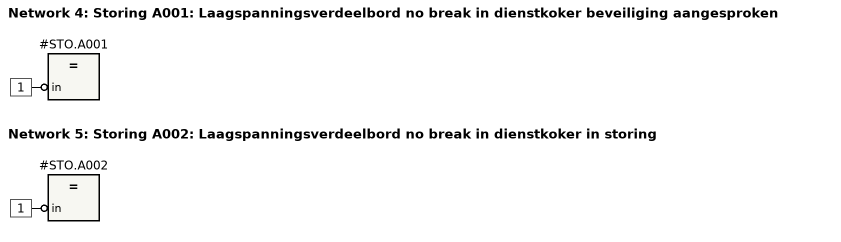
   #STO.A001 := NOT 1;
END_REGION

REGION Network 5: Storing A002: Laagspanningsverdeelbord no break in dienstkoker in storing
   #STO.A002 := NOT 1;
END_REGION

REGION Network 6 (SCL): EINDE
   // Variabelen van intern scada rakvlak naar outputs copieren
   #VAR_IF_OVN.SCL1 := #VAR.SCL1;
   #VAR_IF_OVN.SCL2 := #VAR.SCL2;
   #VAR_IF_OVN.BEV := #VAR.BEV;
END_REGION
END_FUNCTION_BLOCK

FUNCTION_BLOCK "TYPIC_C105_IF_UPS"   // FB23, FBD
TITLE = TYPIC_C105_IF_UPS: No Break
{ S7_Optimized_Access := 'TRUE' }
AUTHOR : OCOTECH
FAMILY : Typical
NAME : C105.701
// Logisch Object Besturing: C105.601
// 
// De interne functie UPS verzorgt de bewaking van een Noobreak installatie.
// stored: MemoryReserve 10, SetENOAutomatically false
   VAR_INPUT
      IN_STS { ExternalAccessible := 'False'; ExternalVisible := 'False'; ExternalWritable := 'False'} : Bool;   // Status van UPS (Batterij / Werking / Bypass)
      IN_TYD { ExternalAccessible := 'False'; ExternalVisible := 'False'; ExternalWritable := 'False'} : Time;   // Resterende autonomietijd (min)
      IN_PWR { ExternalAccessible := 'False'; ExternalVisible := 'False'; ExternalWritable := 'False'} : Real;   // Resterend vermogen
      IN_SPA1 { ExternalAccessible := 'False'; ExternalVisible := 'False'; ExternalWritable := 'False'} : Real;   // Uitgangsspanning 1
      IN_SPA2 { ExternalAccessible := 'False'; ExternalVisible := 'False'; ExternalWritable := 'False'} : Real;   // Uitgangsspanning 2
      IN_SPA3 { ExternalAccessible := 'False'; ExternalVisible := 'False'; ExternalWritable := 'False'} : Real;   // Uitgangsspanning 3
      IN_STR1 { ExternalAccessible := 'False'; ExternalVisible := 'False'; ExternalWritable := 'False'} : Real;   // Uitgangsstroom 1
      IN_STR2 { ExternalAccessible := 'False'; ExternalVisible := 'False'; ExternalWritable := 'False'} : Real;   // Uitgangsstroom 2
      IN_STR3 { ExternalAccessible := 'False'; ExternalVisible := 'False'; ExternalWritable := 'False'} : Real;   // Uitgangsstroom 3
   END_VAR
   VAR_OUTPUT
      VAR_IF_UPS { ExternalAccessible := 'False'; ExternalVisible := 'False'; ExternalWritable := 'False'} : "C105_VAR_IF_UPS_TYPIC";   // Struct met alle variabelen naar bovenliggende functies
   END_VAR
   VAR
      STO { ExternalWritable := 'False'} : Struct   // Storingen
         A001 { ExternalAccessible := 'False'; ExternalVisible := 'False'} : Bool;   // No Break installatie in bypass
         A002 { ExternalAccessible := 'False'; ExternalVisible := 'False'} : Bool;   // No Break installatie uit bedrijf
      END_STRUCT;
      VAR { ExternalWritable := 'False'} : Struct   // Variabelen
         STS1 { ExternalAccessible := 'False'; ExternalVisible := 'False'} : Bool;   // Status UPS [In batterijwerking]
         STS2 { ExternalAccessible := 'False'; ExternalVisible := 'False'} : Bool;   // Status UPS [In bypass]
         STS3 { ExternalAccessible := 'False'; ExternalVisible := 'False'} : Bool;   // Status UPS [In normale werking]
         TYD { ExternalAccessible := 'False'; ExternalVisible := 'False'} : Time;   // Resterende autonomietijd [min]
         PWR { ExternalAccessible := 'False'; ExternalVisible := 'False'} : Real;   // Resterend vermogen
         SPA1 { ExternalAccessible := 'False'; ExternalVisible := 'False'} : Real;   // Uitgangsspanning 1
         SPA2 { ExternalAccessible := 'False'; ExternalVisible := 'False'} : Real;   // Uitgangsspanning 2
         SPA3 { ExternalAccessible := 'False'; ExternalVisible := 'False'} : Real;   // Uitgangsspanning 3
         STR1 { ExternalAccessible := 'False'; ExternalVisible := 'False'} : Real;   // Uitgangsstroom 1
         STR2 { ExternalAccessible := 'False'; ExternalVisible := 'False'} : Real;   // Uitgangsstroom 2
         STR3 { ExternalAccessible := 'False'; ExternalVisible := 'False'} : Real;   // Uitgangsstroom 3
      END_STRUCT;
   END_VAR
BEGIN

REGION Network 1: START
END_REGION

REGION Network 2: +++ Verwerking meetwaarden en statussen +++
   // De meetwaarde en status wordt ontvangen vanuit de interne sturing.
END_REGION

REGION Network 3: +++ Storingen +++
   // Storingen van het systeem
END_REGION

REGION Network 4: Storing A001: No Break installatie in bypass
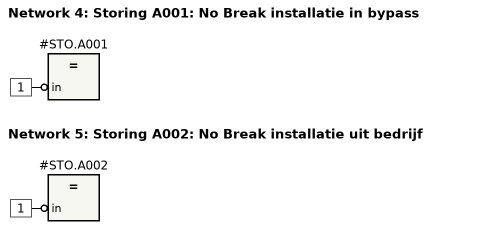
   #STO.A001 := NOT 1;
END_REGION

REGION Network 5: Storing A002: No Break installatie uit bedrijf
   #STO.A002 := NOT 1;
END_REGION

REGION Network 6 (SCL): EINDE
   // Variabelen van intern scada rakvlak naar outputs copieren
   #VAR_IF_UPS.STS1 := #VAR.STS1;
   #VAR_IF_UPS.STS2 := #VAR.STS2;
   #VAR_IF_UPS.STS3 := #VAR.STS3;
   #VAR_IF_UPS.TYD := #VAR.TYD;
   #VAR_IF_UPS.PWR := #VAR.PWR;
   #VAR_IF_UPS.SPA1 := #VAR.SPA1;
   #VAR_IF_UPS.SPA2 := #VAR.SPA2;
   #VAR_IF_UPS.SPA3 := #VAR.SPA3;
   #VAR_IF_UPS.STR1 := #VAR.STR1;
   #VAR_IF_UPS.STR2 := #VAR.STR2;
   #VAR_IF_UPS.STR3 := #VAR.STR3;
END_REGION
END_FUNCTION_BLOCK

FUNCTION_BLOCK "TYPIC_C205_IF_CVE"   // FB26, FBD
{ S7_Optimized_Access := 'TRUE' }
AUTHOR : OCOTECH
FAMILY : Typical
NAME : C205.702
// stored: MemoryReserve 10, SetENOAutomatically false
   VAR_INPUT
      EXT_AUT { ExternalAccessible := 'False'; ExternalVisible := 'False'; ExternalWritable := 'False'} : Bool;   // Externe (hoofd) beveiliging (1 = OK)
      EXT_HW { ExternalAccessible := 'False'; ExternalVisible := 'False'; ExternalWritable := 'False'} : Bool;   // Sturings hardware (PLC) bewaking (1 = OK)
      IN_AUT_C205 { ExternalAccessible := 'False'; ExternalVisible := 'False'; ExternalWritable := 'False'} : Bool;   // Beveiligingen: serie geschakelde terugmelding (1 = OK)
      IN_BAT { ExternalAccessible := 'False'; ExternalVisible := 'False'; ExternalWritable := 'False'} : Bool;   // Batterij (1 = OK)
   END_VAR
   VAR_OUTPUT
      VAR_IF_CVE { ExternalAccessible := 'False'; ExternalVisible := 'False'; ExternalWritable := 'False'} : "C205_VAR_IF_CVE_TYPIC";   // Struct met alle variabelen naar bovenliggende functies
   END_VAR
   VAR
      STO { ExternalWritable := 'False'} : Struct   // Storingen
         A001 : Bool;   // Beveiliging aangesproken
         A002 : Bool;   // Storing batterij
      END_STRUCT;
      VAR { ExternalWritable := 'False'} : Struct   // Variabelen
         EXT_AUT { ExternalAccessible := 'False'; ExternalVisible := 'False'} : Bool;   // Externe (hoofd) beveiliging aangesproken
         EXT_HW { ExternalAccessible := 'False'; ExternalVisible := 'False'} : Bool;   // Sturings hardware (PLC) in storing
      END_STRUCT;
   END_VAR
BEGIN
END_FUNCTION_BLOCK

FUNCTION_BLOCK "TYPIC_C301_BF_VEN"   // FB2, FBD
TITLE = TYPIC_C301_BF_VEN: Ventilatie verkeerskoker
{ S7_Optimized_Access := 'TRUE' }
AUTHOR : OCOTECH
FAMILY : Typical
NAME : C301.801
// Logisch Object Besturing: C301.801
// 
// Het doel van de BF ventilatie is de algemene opvolging, sturing en bediening van de ventilatie van een verkeerskoker.
// stored: MemoryReserve 10, SetENOAutomatically false
   VAR_INPUT
      CFG_TST_UTYD { ExternalAccessible := 'False'; ExternalVisible := 'False'; ExternalWritable := 'False'} : Time;   // Maximale transitietijd stand verandering ventilatie (transitiestatus niet bereikt)
      CFG_TST_OK_TYD { ExternalAccessible := 'False'; ExternalVisible := 'False'; ExternalWritable := 'False'} : Time;   // Stabilisatietijd voor de toestand OK (bereikt)
      CFG_ONHD_TYD { ExternalAccessible := 'False'; ExternalVisible := 'False'; ExternalWritable := 'False'} : Time;   // Waarschuwingstijd start automatische onderhoudstesten
      CFG_MAX_NOK1 { ExternalAccessible := 'False'; ExternalVisible := 'False'; ExternalWritable := 'False'} : Int;   // Maximum aantal onbestuurbare ventilatoren voor beschikbaarheidsstatus beschikbaar
      CFG_MAX_NOK2 { ExternalAccessible := 'False'; ExternalVisible := 'False'; ExternalWritable := 'False'} : Int;   // Maximum aantal onbestuurbare ventilatoren voor beschikbaarheidsstatus beperkt beschikbaar
      STU_CMD_AUT { ExternalAccessible := 'False'; ExternalVisible := 'False'; ExternalWritable := 'False'} : USInt;   // Groepscommando: schakel in automatisch
      STU_AUT_CMD { ExternalAccessible := 'False'; ExternalVisible := 'False'; ExternalWritable := 'False'} : USInt;   // Sturing ventilatie algemeen
      STU_AUT_CMD_DIR { ExternalAccessible := 'False'; ExternalVisible := 'False'; ExternalWritable := 'False'} : USInt;   // Sturing richting
      STU_AUT_VGV_BEV { ExternalAccessible := 'False'; ExternalVisible := 'False'; ExternalWritable := 'False'} : USInt;   // Vrijgave ventilator-beveiligingen onbalans en temperatuur
      STU_VGV_ONHD { ExternalAccessible := 'False'; ExternalVisible := 'False'; ExternalWritable := 'False'} : USInt;   // Vrijgave uitvoeren automatische onderhoudstesten
      STU_ALG_LCK_SIG { ExternalAccessible := 'False'; ExternalVisible := 'False'; ExternalWritable := 'False'} : USInt;   // Onderdruk alarmen
      STU_REG_CAPA { ExternalAccessible := 'False'; ExternalVisible := 'False'; ExternalWritable := 'False'} : USInt;   // Gewenste stand ventilatie bij sensorregeling (afkomstig van CF zichthandhaving)
      STU_ENE_VGV_AAN { ExternalAccessible := 'False'; ExternalVisible := 'False'; ExternalWritable := 'False'} : USInt;   // Vrijgeven of verhinderen bijschakelen energieverbruikers (verlichting / ventilatie)
      STU_ENE_MAX_AAN { ExternalAccessible := 'False'; ExternalVisible := 'False'; ExternalWritable := 'False'} : USInt;   // Maximaal toegelaten ventilatiestand
   END_VAR
   VAR_OUTPUT
      STU_CLUST { ExternalAccessible := 'False'; ExternalVisible := 'False'; ExternalWritable := 'False'} : "C301_STU_CLUST_TYPIC";   // Groepscommando met sturingen naar alle clusters van de ventilatiezone
      VAR_PWR { ExternalAccessible := 'False'; ExternalVisible := 'False'; ExternalWritable := 'False'} : Real;   // Som actueel vermogen van alle clusters
      VAR_CAPA { ExternalAccessible := 'False'; ExternalVisible := 'False'; ExternalWritable := 'False'} : USInt;   // De ingestelde ventilatiestand
      VAR_DIR { ExternalAccessible := 'False'; ExternalVisible := 'False'; ExternalWritable := 'False'} : USInt;   // De ingestelde ventilatierichting
   END_VAR
   VAR_IN_OUT
      CFG_CAPA_DIR1 : Array[1..8] of USInt;   // Omzetting ventilatiestand naar aantal ventilatoren, per cluster (zie verder), rijrichting
      CFG_CAPA_DIR2 : Array[1..8] of USInt;   // Omzetting ventilatiestand naar aantal ventilatoren, per cluster (zie verder), tegenrijrichting
      VAR_CLUST : Array[*] of "C301_VAR_CLUST_TYPIC";   // Array met alle clusters, met alle variabelen van de cluster
   END_VAR
   VAR
      BED : Struct   // Bedieningen
         ALG : Struct   // Gewenste stand
            X : "UDT_BED_ALG";
            KNOP { S7_SetPoint := 'True'} : Array[0..10] of "UDT_BED_KNOP";
         END_STRUCT;
         ALG_DIR : Struct   // Gewenste richting
            X : "UDT_BED_ALG";
            KNOP { S7_SetPoint := 'True'} : Array[0..2] of "UDT_BED_KNOP";
         END_STRUCT;
         VGV_BEV : Struct   // Vrijgave ventilator-beveiligingen onbalans en temperatuur
            X : "UDT_BED_ALG";
            KNOP { S7_SetPoint := 'True'} : Array[0..2] of "UDT_BED_KNOP";
         END_STRUCT;
         ONHD : Struct   // Uitvoeren automatische onderhoudstesten
            X : "UDT_BED_ALG";
            KNOP { S7_SetPoint := 'True'} : Array[0..1] of "UDT_BED_KNOP";
         END_STRUCT;
      END_STRUCT;
      BED_ALG { ExternalWritable := 'False'} : "TYPIC_HF_BED_ALG_KNOP";   // Gewenste stand
      BED_ALG_DIR { ExternalWritable := 'False'} : "TYPIC_HF_BED_ALG_KNOP";   // Gewenste richting
      BED_VGV_BEV { ExternalWritable := 'False'} : "TYPIC_HF_BED_ALG_KNOP";   // Vrijgave ventilator-beveiligingen onbalans en temperatuur
      BED_ONHD { ExternalWritable := 'False'} : "TYPIC_HF_BED_ALG_KNOP";   // Uitvoeren automatische onderhoudstesten
      SIG { ExternalWritable := 'False'} : Struct   // Signaleringen
         AA01 : Bool;   // Gewenste stand niet bereikt
         AA02 : Bool;   // Automatische onderhoudstesten ventilatie
         AB01 : Bool;   // Ventilatie niet beschikbaar
         AB02 : Bool;   // Ventilatie beperkt beschikbaar
      END_STRUCT;
      VAR { ExternalWritable := 'False'} : Struct   // Variabelen
         AUT_SWA : USInt;   // De stand die de ventilatie moet handhaven als de bedieningswijze is ingesteld op automatisch
         REG_CAPA : USInt;   // De stand die de ventilatie moet handhaven als de sensorregeling actief is. Deze waarde wordt bepaald door de coordinerende functie Zichthandhaving Verkeerskoker
         BMO : USInt;   // Bedieningsmode
         AUT_DIR : USInt;   // De richting die de ventilatoren op moeten blazen als de bedieningswijze is ingesteld op automatisch
         DIR_BWA : USInt;   // De werkelijke ventilatierichting
         NIV_BWA : USInt;   // Momentane ventilatieniveau (percentage)
         NIV_AAN_BWA { ExternalAccessible := 'False'; ExternalVisible := 'False'} : USInt;   // Momentaan aantal aangeschakelde ventilatoren
         NIV_AAN_SWA { ExternalAccessible := 'False'; ExternalVisible := 'False'} : USInt;   // Gewenst aantal aangeschakelde ventilatoren
         CAPA_MAX { ExternalAccessible := 'False'; ExternalVisible := 'False'} : USInt;   // Totaal aantal ventilatoren in de ventilatiezone
         CAPA_OK_BWA { ExternalAccessible := 'False'; ExternalVisible := 'False'} : USInt;   // Aantal beschikbare ventilatoren
         CAPA_BWA : USInt;   // De totaal beschikbare ventilatiecapaciteit.
         TST_BWA : USInt;   // De status van de transitie van de langsventilatie
         BSC : USInt;   // Geeft de beschikbaarheid van de langsventilatie aan
         VGV_SIG_VOP : USInt;   // TRUE = Signaleringen vrijgegeven voor verkeersoperator FALSE = Onderdrukt
         ONHD_STS : USInt;   // Status automatische onderhoudstesten
         ONHD_CLUST : USInt;   // Nummer van de cluster die onderhoudstesten dient uit te voeren
         VGV_BEV : USInt;   // Vrijgave ventilator-beveiligingen onbalans en temperatuur
         CAPA : USInt;   // De ingestelde ventilatiestand
         DIR : USInt;   // De ingestelde ventilatierichting
      END_STRUCT;
      HF_TST { ExternalAccessible := 'False'; ExternalVisible := 'False'; ExternalWritable := 'False'} : "TYPIC_HF_TST";   // Hulpfunctie transitiestatus
   END_VAR
   // // BED.ALG.KNOP[0] : Auto
   // // BED.ALG.KNOP[1] : 0 (Uit)
   // // BED.ALG.KNOP[2] : 1
   // // BED.ALG.KNOP[3] : 2
   // // BED.ALG.KNOP[4] : 3
   // // BED.ALG.KNOP[5] : 4
   // // BED.ALG.KNOP[6] : 5
   // // BED.ALG.KNOP[7] : 6
   // // BED.ALG.KNOP[8] : 7
   // // BED.ALG.KNOP[9] : 8
   // // BED.ALG.KNOP[10] : Sensorregeling
   // // BED.ALG_DIR.KNOP[0] : Auto
   // // BED.ALG_DIR.KNOP[1] : Rijrichting
   // // BED.ALG_DIR.KNOP[2] : Tegenrij
   // // BED.VGV_BEV.KNOP[0] : Auto
   // // BED.VGV_BEV.KNOP[1] : Ja
   // // BED.VGV_BEV.KNOP[2] : Onderdrukt
   // // BED.ONHD.KNOP[0] : Aan
   // // BED.ONHD.KNOP[1] : Uit
BEGIN

REGION Network 1: START
END_REGION

REGION Network 2: +++ Bedieningen +++
   // Vrijgave en verwerking van de bedieningen (centrale en lokale bediening). De bedienwaardes worden daarna in de verdere deelfunctionaliteiten gebruikt.
END_REGION

REGION Network 3: Knoppen BED_ALG(Gewenste stand)
   // Waardes en vrijge van de knoppen BED_ALG
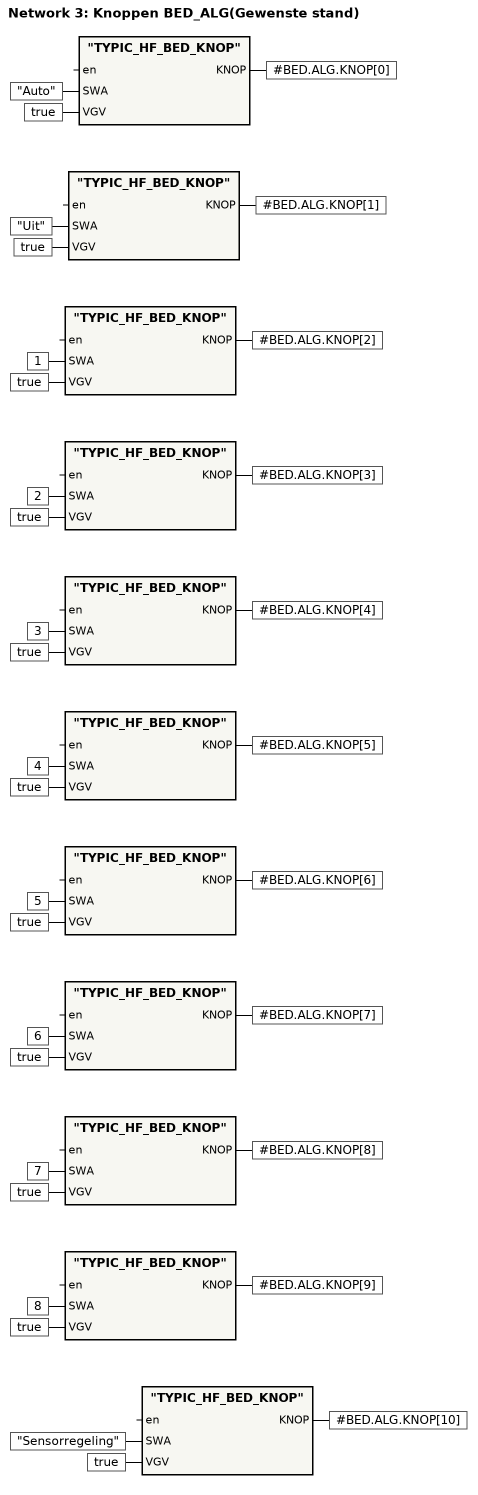
   "TYPIC_HF_BED_KNOP"(SWA := "Auto", VGV := true, KNOP => #BED.ALG.KNOP[0]);
   "TYPIC_HF_BED_KNOP"(SWA := "Uit", VGV := true, KNOP => #BED.ALG.KNOP[1]);
   "TYPIC_HF_BED_KNOP"(SWA := 1, VGV := true, KNOP => #BED.ALG.KNOP[2]);
   "TYPIC_HF_BED_KNOP"(SWA := 2, VGV := true, KNOP => #BED.ALG.KNOP[3]);
   "TYPIC_HF_BED_KNOP"(SWA := 3, VGV := true, KNOP => #BED.ALG.KNOP[4]);
   "TYPIC_HF_BED_KNOP"(SWA := 4, VGV := true, KNOP => #BED.ALG.KNOP[5]);
   "TYPIC_HF_BED_KNOP"(SWA := 5, VGV := true, KNOP => #BED.ALG.KNOP[6]);
   "TYPIC_HF_BED_KNOP"(SWA := 6, VGV := true, KNOP => #BED.ALG.KNOP[7]);
   "TYPIC_HF_BED_KNOP"(SWA := 7, VGV := true, KNOP => #BED.ALG.KNOP[8]);
   "TYPIC_HF_BED_KNOP"(SWA := 8, VGV := true, KNOP => #BED.ALG.KNOP[9]);
   "TYPIC_HF_BED_KNOP"(SWA := "Sensorregeling", VGV := true, KNOP => #BED.ALG.KNOP[10]);
END_REGION

REGION Network 4: BED_ALG(Gewenste stand)
   // Verwerking BED_ALG
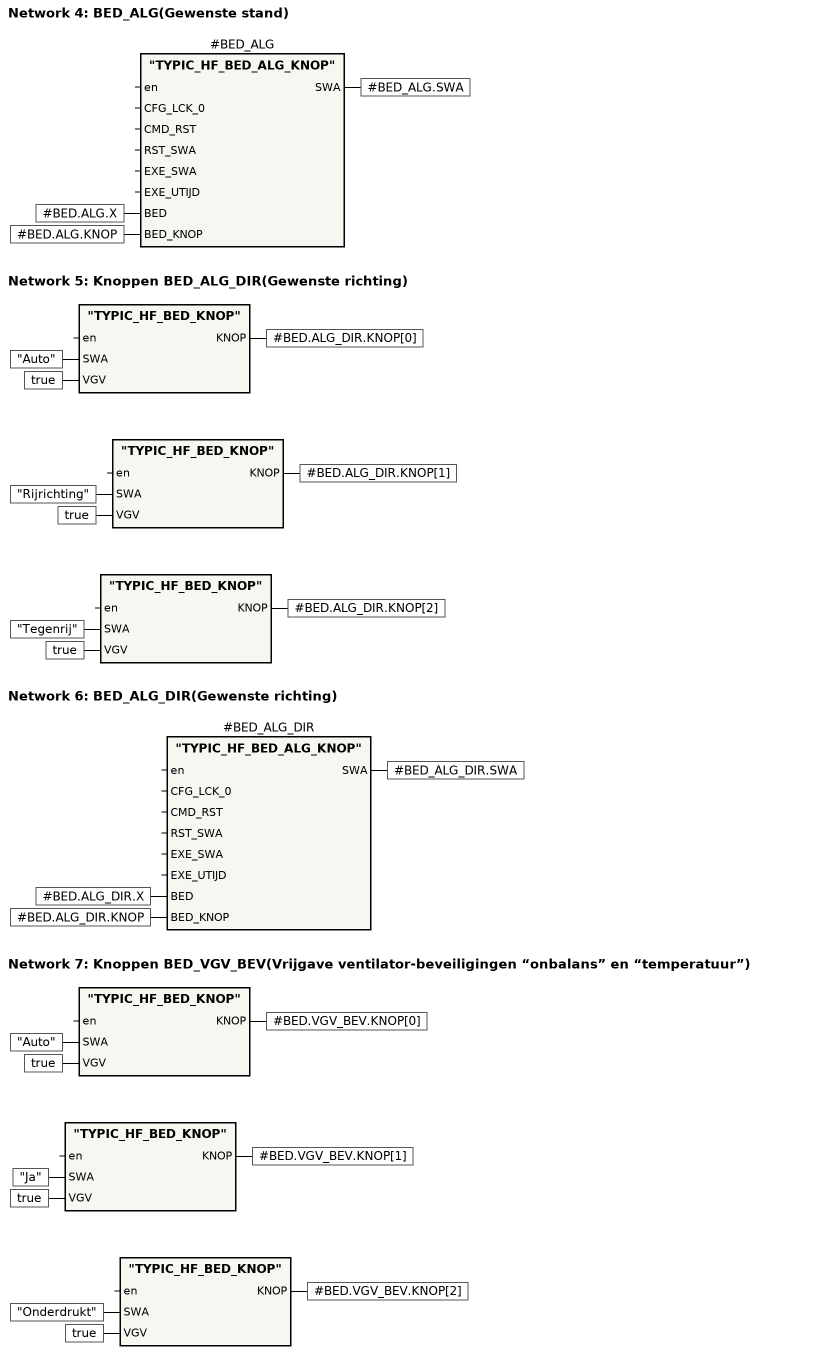
   #BED_ALG(BED := #BED.ALG.X, BED_KNOP := #BED.ALG.KNOP, SWA => #BED_ALG.SWA);   // "TYPIC_HF_BED_ALG_KNOP"
END_REGION

REGION Network 5: Knoppen BED_ALG_DIR(Gewenste richting)
   // Waardes en vrijge van de knoppen BED_ALG_DIR
   "TYPIC_HF_BED_KNOP"(SWA := "Auto", VGV := true, KNOP => #BED.ALG_DIR.KNOP[0]);
   "TYPIC_HF_BED_KNOP"(SWA := "Rijrichting", VGV := true, KNOP => #BED.ALG_DIR.KNOP[1]);
   "TYPIC_HF_BED_KNOP"(SWA := "Tegenrij", VGV := true, KNOP => #BED.ALG_DIR.KNOP[2]);
END_REGION

REGION Network 6: BED_ALG_DIR(Gewenste richting)
   // Verwerking BED_ALG_DIR
   #BED_ALG_DIR(BED := #BED.ALG_DIR.X, BED_KNOP := #BED.ALG_DIR.KNOP, SWA => #BED_ALG_DIR.SWA);   // "TYPIC_HF_BED_ALG_KNOP"
END_REGION

REGION Network 7: Knoppen BED_VGV_BEV(Vrijgave ventilator-beveiligingen “onbalans” en “temperatuur”)
   // Waardes en vrijge van de knoppen BED_VGV_BEV
   "TYPIC_HF_BED_KNOP"(SWA := "Auto", VGV := true, KNOP => #BED.VGV_BEV.KNOP[0]);
   "TYPIC_HF_BED_KNOP"(SWA := "Ja", VGV := true, KNOP => #BED.VGV_BEV.KNOP[1]);
   "TYPIC_HF_BED_KNOP"(SWA := "Onderdrukt", VGV := true, KNOP => #BED.VGV_BEV.KNOP[2]);
END_REGION

REGION Network 8: BED_VGV_BEV(Vrijgave ventilator-beveiligingen “onbalans” en “temperatuur”)
   // Verwerking BED_VGV_BEV
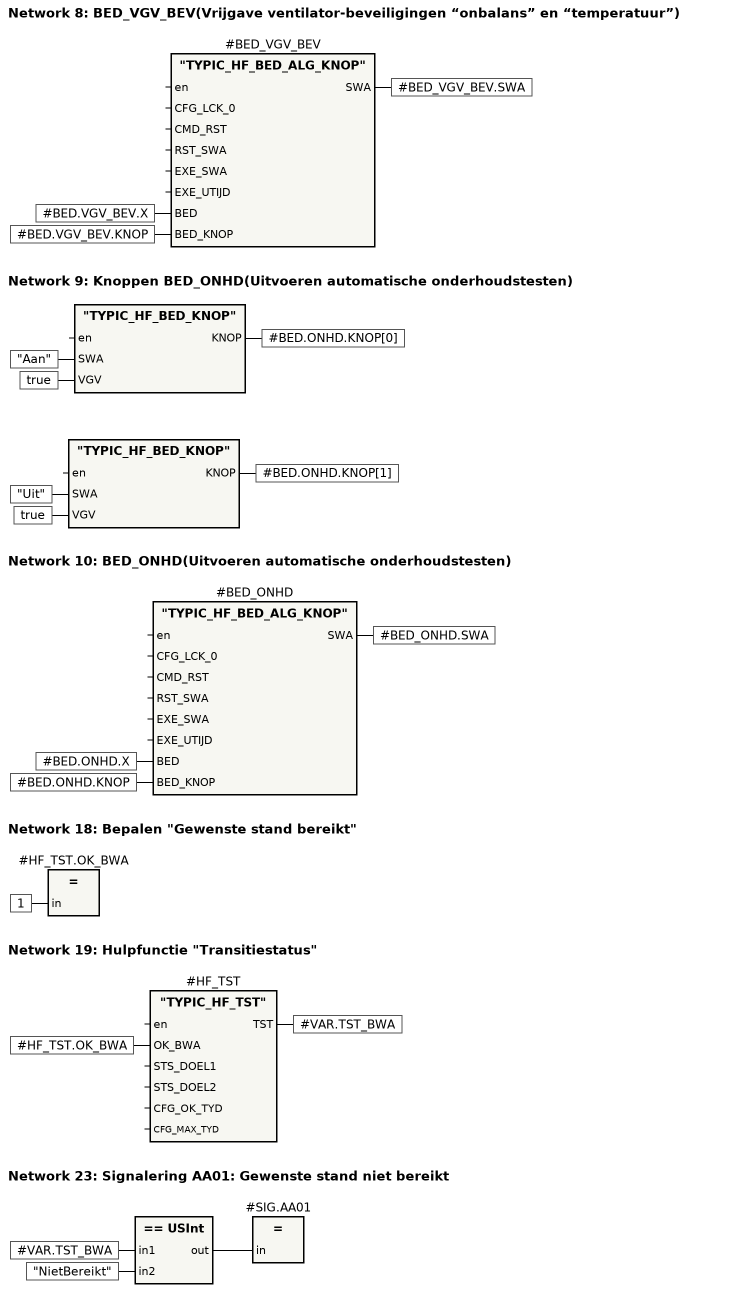
   #BED_VGV_BEV(BED := #BED.VGV_BEV.X, BED_KNOP := #BED.VGV_BEV.KNOP, SWA => #BED_VGV_BEV.SWA);   // "TYPIC_HF_BED_ALG_KNOP"
END_REGION

REGION Network 9: Knoppen BED_ONHD(Uitvoeren automatische onderhoudstesten)
   // Waardes en vrijge van de knoppen BED_ONHD
   "TYPIC_HF_BED_KNOP"(SWA := "Aan", VGV := true, KNOP => #BED.ONHD.KNOP[0]);
   "TYPIC_HF_BED_KNOP"(SWA := "Uit", VGV := true, KNOP => #BED.ONHD.KNOP[1]);
END_REGION

REGION Network 10: BED_ONHD(Uitvoeren automatische onderhoudstesten)
   // Verwerking BED_ONHD
   #BED_ONHD(BED := #BED.ONHD.X, BED_KNOP := #BED.ONHD.KNOP, SWA => #BED_ONHD.SWA);   // "TYPIC_HF_BED_ALG_KNOP"
END_REGION

REGION Network 11: +++ Bepalen bedieningsmode +++
   // Bedieningsmode (Auto / Manueel ) bepalen.
END_REGION

REGION Network 12: +++ Bepalen gewenste capaciteitsinstelling +++
   // Bepalen van de gewenste stand (0..8).
END_REGION

REGION Network 13: +++ Bepalen gewenste ventilatierichting +++
   // Bepalen van de gewenste draairichting (Rijrichting / Tegenrij).
END_REGION

REGION Network 14: +++ Bepalen vrijgave ventilatorbeveiligingen +++
   // Bepalen vrijgave of onderdrukken van de ventilatorbeveiligingen onbalans en temperatuur.
END_REGION

REGION Network 15: +++ Bepalen werkelijke ventilatierichting +++
   // Bepalen van de werkelijke ventilatierichting (Rijrichting / Tegenrij / Onbepaald) aan de hand van de ventilatierichtingen van de ventilatieclusters.
END_REGION

REGION Network 16: +++ Berekeningen +++
   // Verscheidene berekeningen die nodig zijn voor de functionele werking of info voor weergave via de centrale en lokale bediening, zoals het momentane ventilatieniveau, aantal beschikbare ventilatoren, beschikbare capaciteit, actueel vermogen ventilatiezone.
END_REGION

REGION Network 17: +++ Bepalen transitiestatus +++
   // Transitiestatus (bereikt / niet bereikt / in transitie) bepalen.
END_REGION

REGION Network 18: Bepalen "Gewenste stand bereikt"
   // Bepalen of de actuele stand in overeenstemming is met de gewenste stand
   #HF_TST.OK_BWA := 1;
END_REGION

REGION Network 19: Hulpfunctie "Transitiestatus"
   // De transitiestatus geeft de relatie tussen een gewenste stand (van een functionaliteit) en de actuele stand aan.
   #HF_TST(OK_BWA := #HF_TST.OK_BWA, TST => #VAR.TST_BWA);   // "TYPIC_HF_TST"
END_REGION

REGION Network 20: +++ Bepalen beschikbaarheidsstatus +++
   // Beschikbaarheidsstatus (beschikbaar / beperkt beschikbaar / niet beschikbaar) bepalen.
END_REGION

REGION Network 21 (SCL): Beschikbaarheidsstatus bepalen
   IF 
       //voorwaarden "Niet beschikbaar"
       TRUE
   THEN
       //Beschikbaarheidsstatus = Niet Beschikbaar
       #VAR.BSC:= "NietBeschikbaar";
   ELSIF
       //voorwaarden "Beperkt beschikbaar"
       TRUE
   THEN
       //Beschikbaarheidsstatus = Beperkt Beschikbaar
       #VAR.BSC:= "Beperkt";
   ELSE
       //Beschikbaarheidsstatus = Beschikbaar
       #VAR.BSC:= "Beschikbaar";
   END_IF;
END_REGION

REGION Network 22: +++ Signaleringen +++
   // Aanmaken signaleringen.
END_REGION

REGION Network 23: Signalering AA01: Gewenste stand niet bereikt
   #SIG.AA01 := #VAR.TST_BWA = "NietBereikt";
END_REGION

REGION Network 24: Signalering AB01 : Niet Beschikbaar
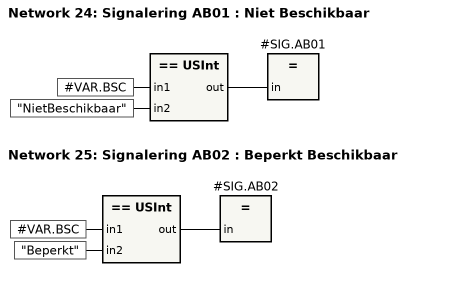
   #SIG.AB01 := #VAR.BSC = "NietBeschikbaar";
END_REGION

REGION Network 25: Signalering AB02 : Beperkt Beschikbaar
   #SIG.AB02 := #VAR.BSC = "Beperkt";
END_REGION

REGION Network 26: +++ Automatische onderhoudstesten +++
   // Functionaliteit waarbij iedere ventilator een voor een aangestuurd wordt ter controle van de goede werking van iedere ventilator.
END_REGION

REGION Network 27: +++ Sturingen +++
   // Uitgeven van sturingen naar de ventilatieclusters.
END_REGION

REGION Network 28: EINDE
   // Variabelen van intern scada rakvlak naar outputs copieren
END_REGION
END_FUNCTION_BLOCK

FUNCTION_BLOCK "TYPIC_C301_IF_VEN"   // FB5, FBD
TITLE = TYPIC_C301_IF_VEN: Ventilator
{ S7_Optimized_Access := 'TRUE' }
AUTHOR : OCOTECH
FAMILY : Typical
NAME : C301.701
// Logisch Object Besturing: C301.701
// 
// De interne functie ventilator verzorgt de interne besturing, bewaking en fysieke aansturing van een aan/uit ventilator.
// 
// Een langsventilator heeft 2 mogelijke draairichtingen:
//  Rijrichting
//  Tegenrij
// Een ingangsventilator heeft 1 mogelijke draairichting:
//  Rijrichting
// stored: MemoryReserve 10, SetENOAutomatically false
   VAR_INPUT
      PULS_100ms { ExternalAccessible := 'False'; ExternalVisible := 'False'; ExternalWritable := 'False'} : Bool;   // Puls, 1 PLC-cyclus hoog, 1 keer per 100 ms
      PULS_1s { ExternalAccessible := 'False'; ExternalVisible := 'False'; ExternalWritable := 'False'} : Bool;   // Puls, 1 PLC-cyclus hoog, 1 keer per seconde
      EXT_AUT { ExternalAccessible := 'False'; ExternalVisible := 'False'; ExternalWritable := 'False'} : Bool;   // Externe (hoofd) beveiliging (1 = OK)
      EXT_HW { ExternalAccessible := 'False'; ExternalVisible := 'False'; ExternalWritable := 'False'} : Bool;   // Sturings hardware (PLC) bewaking (1 = OK)
      IN_HND { ExternalAccessible := 'False'; ExternalVisible := 'False'; ExternalWritable := 'False'} : Bool;   // Terugmelding aansturing via hand (hardware)
      IN_POS { ExternalAccessible := 'False'; ExternalVisible := 'False'; ExternalWritable := 'False'} : Bool;   // Terugmelding aansturing in rijrichting
      IN_NEG { ExternalAccessible := 'False'; ExternalVisible := 'False'; ExternalWritable := 'False'} : Bool;   // Terugmelding aansturing tegenrijrichting
      IN_AUT { ExternalAccessible := 'False'; ExternalVisible := 'False'; ExternalWritable := 'False'} : Bool;   // Status thermische beveiliging (1 = OK)
      IN_PTC { ExternalAccessible := 'False'; ExternalVisible := 'False'; ExternalWritable := 'False'} : Bool;   // Detectie hoge temperatuur in de motorwikkelingen (1 = OK)
      IN_TRL { ExternalAccessible := 'False'; ExternalVisible := 'False'; ExternalWritable := 'False'} : Word;   // Detectie trillingen (onbalans)
      IN_SCW { ExternalAccessible := 'False'; ExternalVisible := 'False'; ExternalWritable := 'False'} : Bool;   // Werkschakelaar (1 = AAN)
      IN_STO { ExternalAccessible := 'False'; ExternalVisible := 'False'; ExternalWritable := 'False'} : Bool;   // Storingsmelding MCC (1 = OK)
      IN_STS1 { ExternalAccessible := 'False'; ExternalVisible := 'False'; ExternalWritable := 'False'} : Bool;   // Status motorlade in (1 = Ingeschakeld )
      IN_STS2 { ExternalAccessible := 'False'; ExternalVisible := 'False'; ExternalWritable := 'False'} : Bool;   // Status motorlade in test (1 = In Test)
      IN_STS3 { ExternalAccessible := 'False'; ExternalVisible := 'False'; ExternalWritable := 'False'} : Bool;   // Status motorlade uitgereden (1 = Uitgereden)
      IN_STR1 { ExternalAccessible := 'False'; ExternalVisible := 'False'; ExternalWritable := 'False'} : Real;   // Analoge meting ventilator fasestroom 1
      IN_STR2 { ExternalAccessible := 'False'; ExternalVisible := 'False'; ExternalWritable := 'False'} : Real;   // Analoge meting ventilator fasestroom 2
      IN_STR3 { ExternalAccessible := 'False'; ExternalVisible := 'False'; ExternalWritable := 'False'} : Real;   // Analoge meting ventilator fasestroom 3
      CFG_2RI { ExternalAccessible := 'False'; ExternalVisible := 'False'; ExternalWritable := 'False'} : Bool;   // TRUE = Ventilator kan in twee richtingen draaien (i.p.v. enkel een richting)
      CFG_UTYD { ExternalAccessible := 'False'; ExternalVisible := 'False'; ExternalWritable := 'False'} : Time;   // Omschakeltijd, tijd die nodig is om uit te bollen in een richting vooraleer de andere richting gestart mag worden.
      CFG_TYD_FB { ExternalAccessible := 'False'; ExternalVisible := 'False'; ExternalWritable := 'False'} : Time;   // Vertragingstijd storing foute terugmelding
      CFG_TYD_TRL { ExternalAccessible := 'False'; ExternalVisible := 'False'; ExternalWritable := 'False'} : Time;   // Vertragingstijd storing onbalans
      CFG_TRL_MAX { ExternalAccessible := 'False'; ExternalVisible := 'False'; ExternalWritable := 'False'} : Real;   // Hoogste waarde scalering trillingsmeting
      CFG_TRL_MIN { ExternalAccessible := 'False'; ExternalVisible := 'False'; ExternalWritable := 'False'} : Real;   // Laagste waarde scalering trillingsmeting
      CFG_TRL_HOOG { ExternalAccessible := 'False'; ExternalVisible := 'False'; ExternalWritable := 'False'} : Real;   // Schakeldrempel hoog trillingsmeting (onbalans)
   END_VAR
   VAR_OUTPUT
      VAR_IF_VEN { ExternalAccessible := 'False'; ExternalVisible := 'False'; ExternalWritable := 'False'} : "C301_VAR_IF_VEN_TYPIC";   // Struct met alle variabelen naar bovenliggende functies
      OUT_POS { ExternalAccessible := 'False'; ExternalVisible := 'False'; ExternalWritable := 'False'} : Bool;   // Aansturen contactor rijrichting
      OUT_NEG { ExternalAccessible := 'False'; ExternalVisible := 'False'; ExternalWritable := 'False'} : Bool;   // Aansturen contactor tegenrij
      OUT_RES { ExternalAccessible := 'False'; ExternalVisible := 'False'; ExternalWritable := 'False'} : Bool;   // Reset van de motorlade storingen
   END_VAR
   VAR_IN_OUT
      STU_IF_VEN : "C301_STU_IF_VEN_TYPIC";   // Struct met alle sturingen van de subfunctie (SF) calamiteitendoorsteek van 3B
      STU_VGV_VEN_AAN : Bool;   // Vrijgave inschakelen
   END_VAR
   VAR
      STO { ExternalWritable := 'False'} : Struct   // Storingen
         A001 : Bool;   // Beveiliging aangesproken
         A002 : Bool;   // Algemene storing MCC
         A003 : Bool;   // Te hoge temperatuur in de wikkelingen van de motor van de ventilator
         A004 : Bool;   // De ventilator is in onbalans
         A005 : Bool;   // Fout stroommeting fase 1
         A006 : Bool;   // Fout stroommeting fase 2
         A007 : Bool;   // Fout stroommeting fase 3
         A008 : Bool;   // Motorlade uitgeschakeld
         A009 : Bool;   // Motorlade in test
         A010 : Bool;   // Motorlade uitgereden
         A011 : Bool;   // Draadbreuk trillingsmeting
         A012 : Bool;   // Meetbereik trillingsmeting overschreden
         AT01 : Bool;   // Discordantie motor: terugmelding niet ontvangen
         AT02 : Bool;   // Discordantie motor: terugmelding blijft aanwezig
         AT03 : Bool;   // Discordantie motor: terugmeldingen Positief en negatief tegelijkertijd
         M001 : Bool;   // Werkschakelaar uitgeschakeld
      END_STRUCT;
      VAR { ExternalWritable := 'False'} : Struct   // Variabelen
         STS_AAN { ExternalAccessible := 'False'; ExternalVisible := 'False'} : Bool;   // TRUE = Ventilator is aangestuurd FALSE = Uit
         DIR_POS { ExternalAccessible := 'False'; ExternalVisible := 'False'} : Bool;   // TRUE = Ventilator draait in positieve richting (rijrichting)
         DIR_NEG { ExternalAccessible := 'False'; ExternalVisible := 'False'} : Bool;   // TRUE = Ventilator draait in negatieve richting (tegenrij)
         BMO_HAND { ExternalAccessible := 'False'; ExternalVisible := 'False'} : Bool;   // TRUE = Ventilator in hand geschakeld FALSE = niet in hand
         TYD_TOT_AAN { ExternalAccessible := 'False'; ExternalVisible := 'False'} : LInt;   // Totaal aantal draaiuren
         TYD_TOT_AAN_UUR { ExternalAccessible := 'False'; ExternalVisible := 'False'} : LInt;   // Totaal aantal draaiuren
         ENE_MWA1 { ExternalAccessible := 'False'; ExternalVisible := 'False'} : Real;   // Stroommeting fase 1
         ENE_MWA2 { ExternalAccessible := 'False'; ExternalVisible := 'False'} : Real;   // Stroommeting fase 2
         ENE_MWA3 { ExternalAccessible := 'False'; ExternalVisible := 'False'} : Real;   // Stroommeting fase 3
         TRL_MWA { ExternalAccessible := 'False'; ExternalVisible := 'False'} : Real;   // Trillingsmeting
         EXT_AUT { ExternalAccessible := 'False'; ExternalVisible := 'False'} : Bool;   // Externe (hoofd) beveiliging aangesproken
         EXT_HW { ExternalAccessible := 'False'; ExternalVisible := 'False'} : Bool;   // Sturings hardware (PLC) in storing
      END_STRUCT;
   END_VAR
BEGIN

REGION Network 1: START
END_REGION

REGION Network 2: +++ Metingen +++
   // Inlezen van de 3 stroommetingen van iedere fase van de motor en inlezen van de trillingsmeting.
END_REGION

REGION Network 3: +++ Storingen +++
   // Verwerken van de storingsmeldingen (inputs).
END_REGION

REGION Network 4: Storing A001: Beveiliging aangesproken
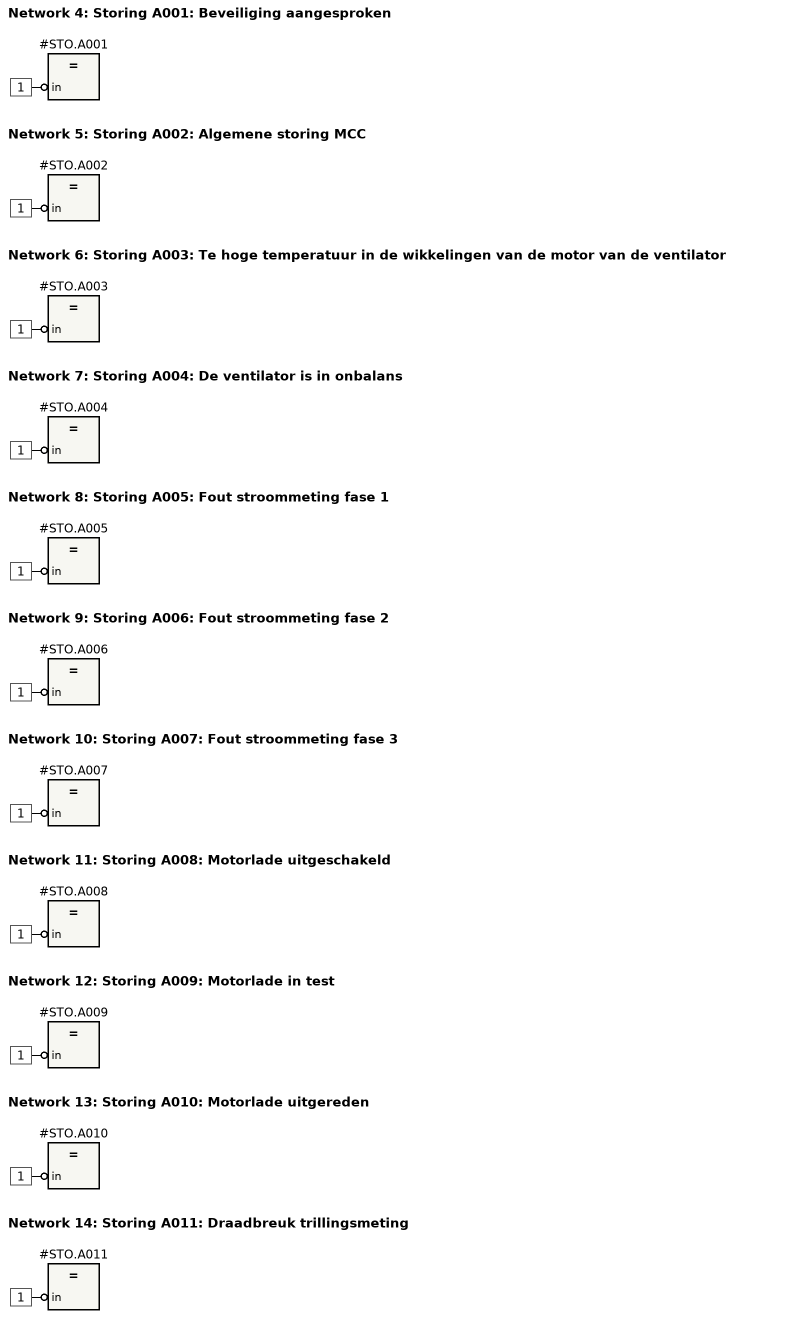
   #STO.A001 := NOT 1;
END_REGION

REGION Network 5: Storing A002: Algemene storing MCC
   #STO.A002 := NOT 1;
END_REGION

REGION Network 6: Storing A003: Te hoge temperatuur in de wikkelingen van de motor van de ventilator
   #STO.A003 := NOT 1;
END_REGION

REGION Network 7: Storing A004: De ventilator is in onbalans
   #STO.A004 := NOT 1;
END_REGION

REGION Network 8: Storing A005: Fout stroommeting fase 1
   #STO.A005 := NOT 1;
END_REGION

REGION Network 9: Storing A006: Fout stroommeting fase 2
   #STO.A006 := NOT 1;
END_REGION

REGION Network 10: Storing A007: Fout stroommeting fase 3
   #STO.A007 := NOT 1;
END_REGION

REGION Network 11: Storing A008: Motorlade uitgeschakeld
   #STO.A008 := NOT 1;
END_REGION

REGION Network 12: Storing A009: Motorlade in test
   #STO.A009 := NOT 1;
END_REGION

REGION Network 13: Storing A010: Motorlade uitgereden
   #STO.A010 := NOT 1;
END_REGION

REGION Network 14: Storing A011: Draadbreuk trillingsmeting
   #STO.A011 := NOT 1;
END_REGION

REGION Network 15: Storing A012: Meetbereik trillingsmeting overschreden
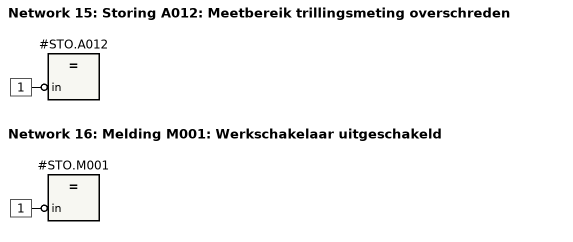
   #STO.A012 := NOT 1;
END_REGION

REGION Network 16: Melding M001: Werkschakelaar uitgeschakeld
   #STO.M001 := NOT 1;
END_REGION

REGION Network 17: +++ Motorsturing +++
   // Aansturen en bewaking van de motor.
END_REGION

REGION Network 18: +++ Urentellers +++
   // Tellen van de tijdsduur dat motor draait of stilstaat.
END_REGION

REGION Network 19 (SCL): EINDE
   // Variabelen van intern scada rakvlak naar outputs copieren
   #VAR_IF_VEN.STS_AAN := #VAR.STS_AAN;
   #VAR_IF_VEN.DIR_POS := #VAR.DIR_POS;
   #VAR_IF_VEN.DIR_NEG := #VAR.DIR_NEG;
   #VAR_IF_VEN.BMO_HAND := #VAR.BMO_HAND;
   #VAR_IF_VEN.TYD_TOT_AAN := #VAR.TYD_TOT_AAN;
   #VAR_IF_VEN.TYD_TOT_AAN_UUR := #VAR.TYD_TOT_AAN_UUR;
   #VAR_IF_VEN.ENE_MWA1 := #VAR.ENE_MWA1;
   #VAR_IF_VEN.ENE_MWA2 := #VAR.ENE_MWA2;
   #VAR_IF_VEN.ENE_MWA3 := #VAR.ENE_MWA3;
   #VAR_IF_VEN.TRL_MWA := #VAR.TRL_MWA;
   #VAR_IF_VEN.EXT_AUT := #VAR.EXT_AUT;
   #VAR_IF_VEN.EXT_HW := #VAR.EXT_HW;
   #VAR_IF_VEN.STO := #STO;
END_REGION
END_FUNCTION_BLOCK

FUNCTION_BLOCK "TYPIC_C301_SF_VEN"   // FB6, FBD
TITLE = TYPIC_C301_SF_VEN: Ventilator verkeerskoker
{ S7_Optimized_Access := 'TRUE' }
AUTHOR : OCOTECH
FAMILY : Typical
NAME : C301.803
// Logisch Object Besturing: C301.803
// 
// De subfunctie “ventilator verkeerskoker” verzorgt de bediening en sturing van een ventilator vanuit 3B en is tevens het raakvlak tussen 3B en de interne sturing van de ventilator.
// 
// De subfunctie kan zowel gebruikt worden voor langsventilatoren als ingangsventilatoren.
// 
// Een langsventilator heeft 2 mogelijke draairichtingen:
//  Rijrichting
//  Tegenrij
// 
// Een ingangsventilator heeft slechts 1 mogelijke draairichting:
//  Rijrichting
// 
// Deze typical werkt op dezelfde manier voor ingangsventilatoren als langsventilatoren. Bij ingangsventilatoren komen in de praktijk een aantal mogelijkheden nooit voor:
//  Op IRIS SCADA is er een andere typical voor ingangsventilatoren, deze typical heeft geen mogelijkheid voor bediening “Tegenrij”
//  Vanuit de basisfunctie wordt een cluster met ingangsventilatoren nooit in “Tegenrij” aangestuurd 
//  De waarde “Tegenrij” is nooit van toepassing voor statussen of sturingen
//  Signaleringen met betrekking tot “Tegenrij” komen nooit op
// stored: MemoryReserve 10, SetENOAutomatically false
   VAR_INPUT
      CFG_PWR { ExternalAccessible := 'False'; ExternalVisible := 'False'; ExternalWritable := 'False'} : Real;   // Vermogen ventilator
      CFG_IVEN { ExternalAccessible := 'False'; ExternalVisible := 'False'; ExternalWritable := 'False'} : USInt;   // De ventilator is een ingangsventilator
      STU_CMD_AUT { ExternalAccessible := 'False'; ExternalVisible := 'False'; ExternalWritable := 'False'} : USInt;   // Groepscommando: schakel in automatisch
      STU_ALG_LCK_SIG { ExternalAccessible := 'False'; ExternalVisible := 'False'; ExternalWritable := 'False'} : USInt;   // Onderdruk alarmen
      STU_ENE_VGV_AAN { ExternalAccessible := 'False'; ExternalVisible := 'False'; ExternalWritable := 'False'} : USInt;   // Vrijgeven of verhinderen bijschakelen energieverbruikers (verlichting / ventilatie)
   END_VAR
   VAR_OUTPUT
      VAR_VEN { ExternalAccessible := 'False'; ExternalVisible := 'False'; ExternalWritable := 'False'} : "C301_VAR_VEN_TYPIC";   // Struct met alle variabelen van de ventilator
      STU_IF_VEN { ExternalAccessible := 'False'; ExternalVisible := 'False'; ExternalWritable := 'False'} : "C301_STU_IF_VEN_TYPIC";   // Struct met alle sturingen naar de functie (IF) in de interne sturing van de ventilator
   END_VAR
   VAR_IN_OUT
      CMD : USInt;   // Sturing ventilator
      BST : USInt;   // Sturing In Dienst / Uit Dienst
      VGV_BEV : USInt;   // Vrijgave ventilator-beveiligingen onbalans en temperatuur
   END_VAR
   VAR
      BED : Struct   // Bedieningen
         ALG : Struct   // Gewenste stand
            X : "UDT_BED_ALG";
            KNOP { S7_SetPoint := 'True'} : Array[0..3] of "UDT_BED_KNOP";
         END_STRUCT;
         BST : Struct   // Bestuurbaarheid
            X : "UDT_BED_ALG";
            KNOP { S7_SetPoint := 'True'} : Array[0..1] of "UDT_BED_KNOP";
         END_STRUCT;
         RES : Struct   // Reset Storingen
            X : "UDT_BED_ALG";
            KNOP { S7_SetPoint := 'True'} : Array[0..0] of "UDT_BED_KNOP";
         END_STRUCT;
      END_STRUCT;
      BED_ALG { ExternalWritable := 'False'} : "TYPIC_HF_BED_ALG_KNOP";   // Gewenste stand
      BED_BST { ExternalWritable := 'False'} : "TYPIC_HF_BED_ALG_KNOP";   // Bestuurbaarheid
      BED_RES { ExternalWritable := 'False'} : "TYPIC_HF_BED_ALG_KNOP";   // Reset Storingen
      SIG { ExternalWritable := 'False'} : Struct   // Signaleringen
         AA01 : Bool;   // Ventilator niet bestuurbaar
         AA02 : Bool;   // Ventilator geeft storing, maar is bestuurbaar
         A001 : Bool;   // Beveiliging aangesproken
         A002 : Bool;   // Algemene storing MCC
         A003 : Bool;   // Te hoge temperatuur in de wikkelingen van de motor van de ventilator
         A004 : Bool;   // De ventilator is in onbalans
         A005 : Bool;   // Fout stroommeting fase 1
         A006 : Bool;   // Fout stroommeting fase 2
         A007 : Bool;   // Fout stroommeting fase 3
         A008 : Bool;   // Motorlade uitgeschakeld
         A009 : Bool;   // Motorlade in test
         A010 : Bool;   // Motorlade uitgereden
         A011 : Bool;   // Draadbreuk trillingsmeting
         A012 : Bool;   // Meetbereik trillingsmeting overschreden
         AT01 : Bool;   // Foute terugmelding: Motor aangestuurd, terugmelding Aan niet (of te laat) ontvangen
         AT02 : Bool;   // Foute terugmelding: Motor niet aangestuurd, terugmelding Aan blijft aanwezig
         AT03 : Bool;   // Foute terugmeldingen: terugmeldingen Positief en negatief tegelijkertijd
         M001 : Bool;   // Werkschakelaar uitgeschakeld
      END_STRUCT;
      VAR { ExternalWritable := 'False'} : Struct   // Variabelen
         TYD_TOT_AAN_UUR : USInt;   // Totaal aantal draaiuren
         ENE_MWA1 : Real;   // Stroommeting fase 1
         ENE_MWA2 : Real;   // Stroommeting fase 2
         ENE_MWA3 : Real;   // Stroommeting fase 3
         TRL_MWA : USInt;   // Trillingsmeting
         RNB : USInt;   // Reden niet bestuurbaar
         AUT : USInt;   // Beveiliging aangesproken
         VGV_SIG_VOP : Bool;   // TRUE = Signaleringen vrijgegeven voor verkeersoperator FALSE = Onderdrukt
         STS : USInt;   // Status van de ventilator
         DIR : USInt;   // Richting van de ventilator
         BMO : USInt;   // Bedieningsmode
         BST { ExternalAccessible := 'False'; ExternalVisible := 'False'} : USInt;   // Bestuurbaarheid
         PWR { ExternalAccessible := 'False'; ExternalVisible := 'False'} : Real;   // Vermogen van de ventilator
         TYD_TOT_AAN { ExternalAccessible := 'False'; ExternalVisible := 'False'} : USInt;   // Totaal aantal draaiuren
      END_STRUCT;
      HF_BST_OBS { ExternalAccessible := 'False'; ExternalVisible := 'False'; ExternalWritable := 'False'} : "TYPIC_HF_BST_OBS";   // Hulp functie besturing
   END_VAR
   // // BED.ALG.KNOP[0] : Auto
   // // BED.ALG.KNOP[1] : Rijrichting
   // // BED.ALG.KNOP[2] : Tegenrij
   // // BED.ALG.KNOP[3] : Uit
   // // BED.BST.KNOP[0] : InDienst
   // // BED.BST.KNOP[1] : UitDienst
   // // BED.RES.KNOP[0] : Reset
BEGIN

REGION Network 1: START
END_REGION

REGION Network 2: +++ Bedieningen +++
   // Vrijgave en verwerking van de bedieningen (centrale en lokale bediening). De bedienwaardes worden daarna in de verdere deelfunctionaliteiten gebruikt.
END_REGION

REGION Network 3: Knoppen BED_ALG(Gewenste stand)
   // Waardes en vrijge van de knoppen BED_ALG
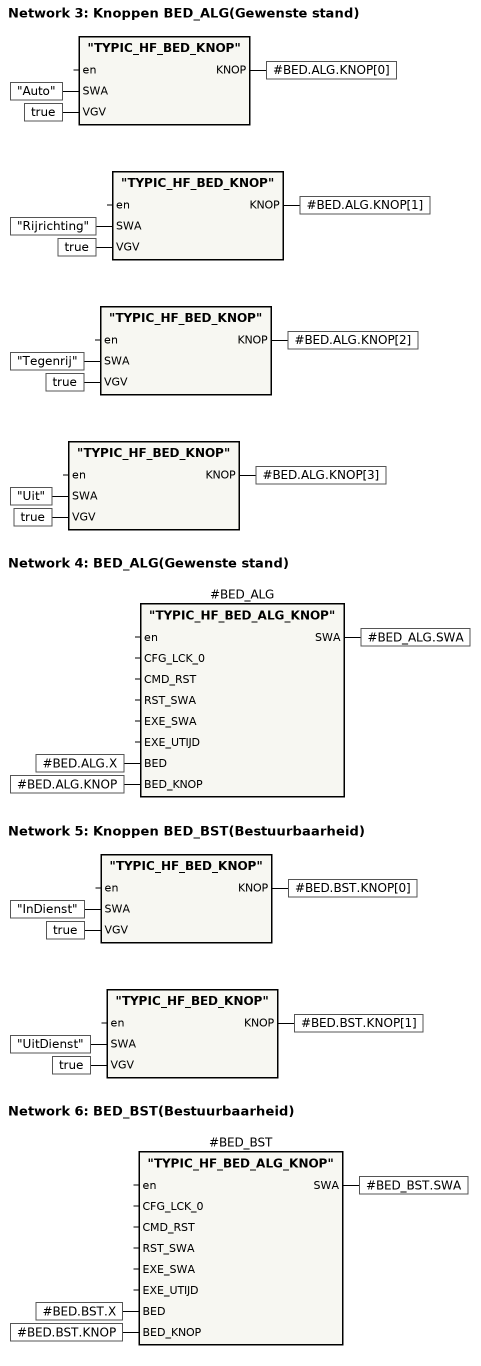
   "TYPIC_HF_BED_KNOP"(SWA := "Auto", VGV := true, KNOP => #BED.ALG.KNOP[0]);
   "TYPIC_HF_BED_KNOP"(SWA := "Rijrichting", VGV := true, KNOP => #BED.ALG.KNOP[1]);
   "TYPIC_HF_BED_KNOP"(SWA := "Tegenrij", VGV := true, KNOP => #BED.ALG.KNOP[2]);
   "TYPIC_HF_BED_KNOP"(SWA := "Uit", VGV := true, KNOP => #BED.ALG.KNOP[3]);
END_REGION

REGION Network 4: BED_ALG(Gewenste stand)
   // Verwerking BED_ALG
   #BED_ALG(BED := #BED.ALG.X, BED_KNOP := #BED.ALG.KNOP, SWA => #BED_ALG.SWA);   // "TYPIC_HF_BED_ALG_KNOP"
END_REGION

REGION Network 5: Knoppen BED_BST(Bestuurbaarheid)
   // Waardes en vrijge van de knoppen BED_BST
   "TYPIC_HF_BED_KNOP"(SWA := "InDienst", VGV := true, KNOP => #BED.BST.KNOP[0]);
   "TYPIC_HF_BED_KNOP"(SWA := "UitDienst", VGV := true, KNOP => #BED.BST.KNOP[1]);
END_REGION

REGION Network 6: BED_BST(Bestuurbaarheid)
   // Verwerking BED_BST
   #BED_BST(BED := #BED.BST.X, BED_KNOP := #BED.BST.KNOP, SWA => #BED_BST.SWA);   // "TYPIC_HF_BED_ALG_KNOP"
END_REGION

REGION Network 7: Knoppen BED_RES(Reset Storingen)
   // Waardes en vrijge van de knoppen BED_RES
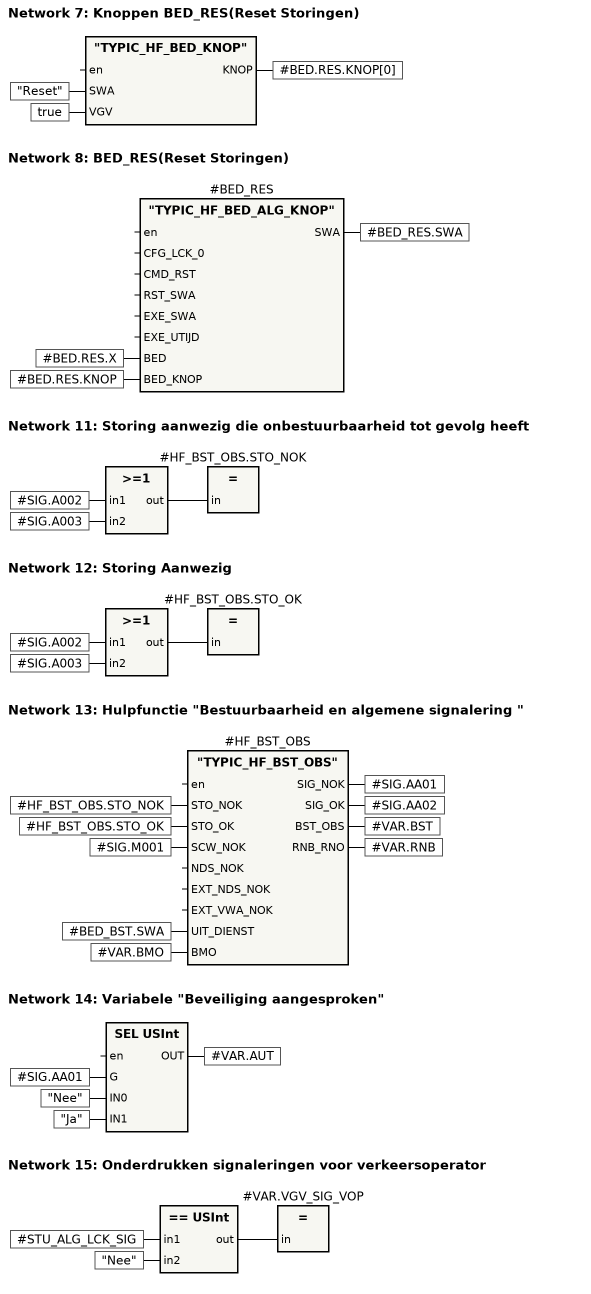
   "TYPIC_HF_BED_KNOP"(SWA := "Reset", VGV := true, KNOP => #BED.RES.KNOP[0]);
END_REGION

REGION Network 8: BED_RES(Reset Storingen)
   // Verwerking BED_RES
   #BED_RES(BED := #BED.RES.X, BED_KNOP := #BED.RES.KNOP, SWA => #BED_RES.SWA);   // "TYPIC_HF_BED_ALG_KNOP"
END_REGION

REGION Network 9: +++ Bepalen bedieningsmode +++
   // Bedieningsmode (Auto / Manueel / Hand) bepalen.
END_REGION

REGION Network 10: +++ Signaleringen en bestuurbaarheid +++
   // Aanmaken signaleringen, bepalen bestuurbaarheid (bestuurbaar / niet bestuurbaar) en bepalen reden van niet bestuurbaarheid.
END_REGION

REGION Network 11: Storing aanwezig die onbestuurbaarheid tot gevolg heeft
   // OR-verknoping van alle storingen om input STO_BST_NOK van de hulpfunctie "Bestuurbaarheid en algemene signlaring"
   #HF_BST_OBS.STO_NOK := #SIG.A002 OR #SIG.A003;
END_REGION

REGION Network 12: Storing Aanwezig
   // OR-verknoping van alle storingen om input STO_BST_OK van de hulpfunctie "Bestuurbaarheid en algemene signlaring"
   #HF_BST_OBS.STO_OK := #SIG.A002 OR #SIG.A003;
END_REGION

REGION Network 13: Hulpfunctie "Bestuurbaarheid en algemene signalering "
   // Bepalen variabele "bestuurbaarheid" en "reden niet bestuurbaar", Signaleringen "bestuurbaarheid" en "algmene storing".
   #HF_BST_OBS(STO_NOK := #HF_BST_OBS.STO_NOK,   // "TYPIC_HF_BST_OBS"
               STO_OK := #HF_BST_OBS.STO_OK,
               SCW_NOK := #SIG.M001,
               UIT_DIENST := #BED_BST.SWA,
               BMO := #VAR.BMO,
               SIG_NOK => #SIG.AA01,
               SIG_OK => #SIG.AA02,
               BST_OBS => #VAR.BST,
               RNB_RNO => #VAR.RNB);
END_REGION

REGION Network 14: Variabele "Beveiliging aangesproken"
   // De variabele VAR_AUT geef aan of er een beveilliging aangesproken is. Deze variabele laat toe dat de verkeersoperator op SCADA kan zien of er een beveilliging aangesproken is voor deze component.
   #VAR.AUT := SEL(G := #SIG.AA01, IN0 := "Nee", IN1 := "Ja");
END_REGION

REGION Network 15: Onderdrukken signaleringen voor verkeersoperator
   // Via de variabele VGV_SIG_VOP wordt aan IRIS SCADA doorgegeven of signaleringen (bestemd voor de verkeersoperator) van de deze functie zichtbaar (of onderdrukt) moeten zijn.
   #VAR.VGV_SIG_VOP := #STU_ALG_LCK_SIG = "Nee";
END_REGION

REGION Network 16: +++ Bepalen status en actueel vermogen +++
   // Status (Aan / Uit) en actueel verbruikt vermogen bepalen.
END_REGION

REGION Network 17: +++ Bepalen actuele ventilatierichting +++
   // De actuele draairichting (Uit / Rijrichting / Tegenrij) bepalen.
END_REGION

REGION Network 18: +++ Draaiuren, fasestromen en trillingsmeting +++
   // Totaal aantal draaiuren, fasestromen en trillingsmeting verwerken.
END_REGION

REGION Network 19: +++ Sturingen +++
   // Commandos naar de interne sturing van de ventilator uitsturen.
END_REGION

REGION Network 20 (SCL): EINDE
   // Variabelen van intern scada rakvlak naar outputs copieren
   #VAR_VEN.STS := #VAR.STS;
   #VAR_VEN.DIR := #VAR.DIR;
   #VAR_VEN.BMO := #VAR.BMO;
   #VAR_VEN.BST := #VAR.BST;
   #VAR_VEN.PWR := #VAR.PWR;
   #VAR_VEN.TYD_TOT_AAN := #VAR.TYD_TOT_AAN;
END_REGION
END_FUNCTION_BLOCK

FUNCTION_BLOCK "TYPIC_C301_SF_VEN_CLUST"   // FB7, FBD
TITLE = TYPIC_C301_SF_VEN_CLUST: Ventilatiecluster verkeerskoker
{ S7_Optimized_Access := 'TRUE' }
AUTHOR : OCOTECH
FAMILY : Typical
NAME : C301.802
// Logisch Object Besturing: C301.802
// 
// Het doel van de SF ventilatiecluster is het aansturen van een cluster van ventilatoren op basis van sturingen ontvangen van de basisfunctie “ventilatie”, bedieningen op IRIS SCADA en de status van de aangestuurde ventilatoren
// stored: MemoryReserve 10, SetENOAutomatically false
   VAR_INPUT
      CFG_NUM { ExternalAccessible := 'False'; ExternalVisible := 'False'; ExternalWritable := 'False'} : USInt;   // Nummer van de cluster binnen ventilatiezone 0 = ingangscluster
      CFG_TYD_ONHD1 { ExternalAccessible := 'False'; ExternalVisible := 'False'; ExternalWritable := 'False'} : USInt;   // Tijdsduur aansturing ventilator bij automatische onderhoudstesten
      CFG_TYD_ONHD2 { ExternalAccessible := 'False'; ExternalVisible := 'False'; ExternalWritable := 'False'} : USInt;   // Tijdsduur intervaltijd bij automatische onderhoudstesten
      STU_CMD_AUT { ExternalAccessible := 'False'; ExternalVisible := 'False'; ExternalWritable := 'False'} : USInt;   // Groepscommando: schakel in automatisch
      STU_ALG_LCK_SIG { ExternalAccessible := 'False'; ExternalVisible := 'False'; ExternalWritable := 'False'} : USInt;   // Onderdruk alarmen
      STU_ENE_VGV_AAN { ExternalAccessible := 'False'; ExternalVisible := 'False'; ExternalWritable := 'False'} : USInt;   // Vrijgeven of verhinderen bijschakelen energieverbruikers (verlichting / ventilatie)
      STU_ENE_MAX_AAN { ExternalAccessible := 'False'; ExternalVisible := 'False'; ExternalWritable := 'False'} : USInt;   // Maximaal toegelaten ventilatiestand
   END_VAR
   VAR_OUTPUT
      VAR_CLUST { ExternalAccessible := 'False'; ExternalVisible := 'False'; ExternalWritable := 'False'} : "C301_VAR_CLUST_TYPIC";   // Struct met alle variabelen van de cluster (info naar de bovenliggende basisfunctie)
      STU_VEN1 { ExternalAccessible := 'False'; ExternalVisible := 'False'; ExternalWritable := 'False'} : "C301_STU_VEN_TYPIC";   // sturing naar ventilator 1
      STU_VEN2 { ExternalAccessible := 'False'; ExternalVisible := 'False'; ExternalWritable := 'False'} : "C301_STU_VEN_TYPIC";   // sturing naar ventilator 2
      STU_VEN3 { ExternalAccessible := 'False'; ExternalVisible := 'False'; ExternalWritable := 'False'} : "C301_STU_VEN_TYPIC";   // sturing naar ventilator 3
      STU_VEN4 { ExternalAccessible := 'False'; ExternalVisible := 'False'; ExternalWritable := 'False'} : "C301_STU_VEN_TYPIC";   // sturing naar ventilator 4
      STU_VEN5 { ExternalAccessible := 'False'; ExternalVisible := 'False'; ExternalWritable := 'False'} : "C301_STU_VEN_TYPIC";   // sturing naar ventilator 5
      STU_VEN6 { ExternalAccessible := 'False'; ExternalVisible := 'False'; ExternalWritable := 'False'} : "C301_STU_VEN_TYPIC";   // sturing naar ventilator 6
      STU_VEN7 { ExternalAccessible := 'False'; ExternalVisible := 'False'; ExternalWritable := 'False'} : "C301_STU_VEN_TYPIC";   // sturing naar ventilator 7
      STU_VEN8 { ExternalAccessible := 'False'; ExternalVisible := 'False'; ExternalWritable := 'False'} : "C301_STU_VEN_TYPIC";   // sturing naar ventilator 8
   END_VAR
   VAR_IN_OUT
      CFG_CAPA_DIR1 : Array[1..8] of USInt;   // Omzetting ventilatiestand naar aantal ventilatoren, per cluster (zie verder), rijrichting
      CFG_CAPA_DIR2 : Array[1..8] of USInt;   // Omzetting ventilatiestand naar aantal ventilatoren, per cluster (zie verder), tegenrijrichting
      VAR_VEN : Array[*] of "C301_VAR_VEN_TYPIC";   // Array met alle ventilatoren, met alle variabelen van de ventilator
      STU_CLUST : "C301_STU_CLUST_TYPIC";   // Struct met alle sturingen vanuit de basisfunctie naar de cluster
   END_VAR
   VAR
      BED : Struct   // Bedieningen
         ALG : Struct   // Gewenste stand
            X : "UDT_BED_ALG";
            KNOP { S7_SetPoint := 'True'} : Array[0..2] of "UDT_BED_KNOP";
         END_STRUCT;
         BST : Struct   // Bestuurbaarheid
            X : "UDT_BED_ALG";
            KNOP { S7_SetPoint := 'True'} : Array[0..1] of "UDT_BED_KNOP";
         END_STRUCT;
      END_STRUCT;
      BED_ALG { ExternalWritable := 'False'} : "TYPIC_HF_BED_ALG_KNOP";   // Gewenste stand
      BED_BST { ExternalWritable := 'False'} : "TYPIC_HF_BED_ALG_KNOP";   // Bestuurbaarheid
      VAR { ExternalWritable := 'False'} : Struct   // Variabelen
         CAPA : USInt;   // Gewenste capaciteitsinstelling
         NIV_SWA { ExternalAccessible := 'False'; ExternalVisible := 'False'} : USInt;   // Gewenst aantal aangeschakelde ventilatoren
         ONHD_VEN { ExternalAccessible := 'False'; ExternalVisible := 'False'} : USInt;   // Nummer ventilator bezig met onderhoudstest
         STU { ExternalAccessible := 'False'; ExternalVisible := 'False'} : USInt;   // Array met de sturingen naar iedere ventilator
         CAPA_OK { ExternalAccessible := 'False'; ExternalVisible := 'False'} : USInt;   // Aantal bestuurbare ventilatoren in de cluster
         NIV_AAN_BWA : USInt;   // Aantal aangeschakelde ventilatoren in de gewenste ventilatierichting
         DIR : USInt;   // Richting van de cluster
         BMO : USInt;   // Bedieningsmode
         ONHD_STS : USInt;   // Status automatische onderhoudstesten
         PWR { ExternalAccessible := 'False'; ExternalVisible := 'False'} : Real;   // Actueel vermogen van de ventilatiecluster
      END_STRUCT;
   END_VAR
   // // BED.ALG.KNOP[0] : Auto
   // // BED.ALG.KNOP[1] : 0 (Uit)
   // // BED.ALG.KNOP[2] : 8
   // // BED.BST.KNOP[0] : InDienst
   // // BED.BST.KNOP[1] : UitDienst
BEGIN

REGION Network 1: START
END_REGION

REGION Network 2: +++ Bedieningen +++
   // Vrijgave en verwerking van de bedieningen (centrale en lokale bediening). De bedienwaardes worden daarna in de verdere deelfunctionaliteiten gebruikt.
END_REGION

REGION Network 3: Knoppen BED_ALG(Gewenste stand)
   // Waardes en vrijge van de knoppen BED_ALG
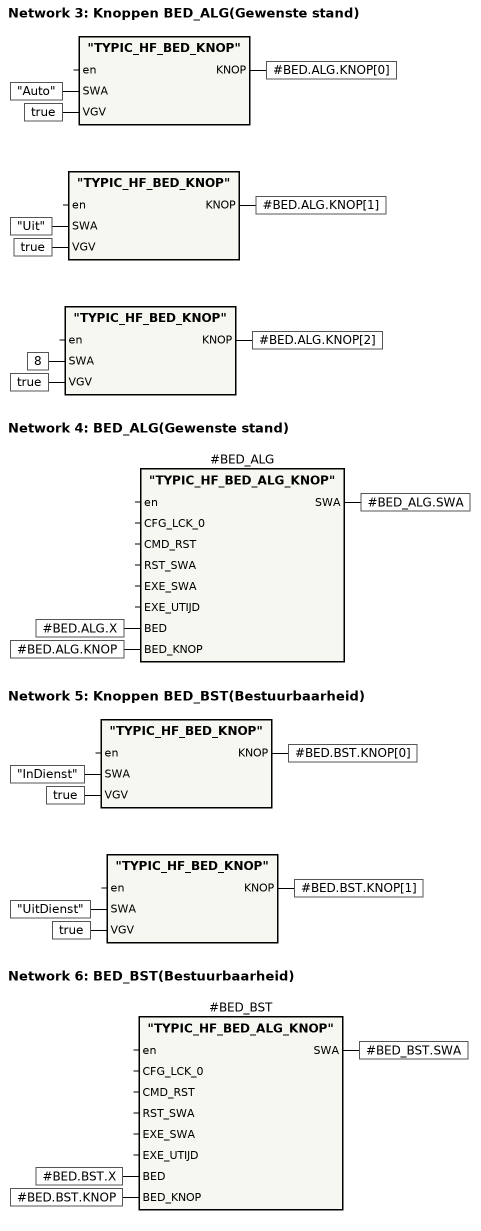
   "TYPIC_HF_BED_KNOP"(SWA := "Auto", VGV := true, KNOP => #BED.ALG.KNOP[0]);
   "TYPIC_HF_BED_KNOP"(SWA := "Uit", VGV := true, KNOP => #BED.ALG.KNOP[1]);
   "TYPIC_HF_BED_KNOP"(SWA := 8, VGV := true, KNOP => #BED.ALG.KNOP[2]);
END_REGION

REGION Network 4: BED_ALG(Gewenste stand)
   // Verwerking BED_ALG
   #BED_ALG(BED := #BED.ALG.X, BED_KNOP := #BED.ALG.KNOP, SWA => #BED_ALG.SWA);   // "TYPIC_HF_BED_ALG_KNOP"
END_REGION

REGION Network 5: Knoppen BED_BST(Bestuurbaarheid)
   // Waardes en vrijge van de knoppen BED_BST
   "TYPIC_HF_BED_KNOP"(SWA := "InDienst", VGV := true, KNOP => #BED.BST.KNOP[0]);
   "TYPIC_HF_BED_KNOP"(SWA := "UitDienst", VGV := true, KNOP => #BED.BST.KNOP[1]);
END_REGION

REGION Network 6: BED_BST(Bestuurbaarheid)
   // Verwerking BED_BST
   #BED_BST(BED := #BED.BST.X, BED_KNOP := #BED.BST.KNOP, SWA => #BED_BST.SWA);   // "TYPIC_HF_BED_ALG_KNOP"
END_REGION

REGION Network 7: +++ Bepalen bedieningsmode en gewenste capaciteitsinstelling +++
   // Bedieningsmode (Auto / Manueel ) bepalen en gewenste stand (0..8) bepalen
END_REGION

REGION Network 8: +++ Bepalen werkelijke ventilatierichting +++
   // Bepalen van de werkelijke ventilatierichting (Rijrichting / Tegenrij / Onbepaald) aan de hand van de ventilatierichtingen van de ventilatieclusters.
END_REGION

REGION Network 9: +++ Bepalen gewenst aantal ventilatoren +++
   // Bepalen van het gewenst aantal ingeschakelde ventilatoren.
END_REGION

REGION Network 10: +++ Bepalen aansturing ventilatoren +++
   // Sturing van iedere individuele ventilator bepalen op basis van de werkingsmode en bestuurbaarheid van de ventilator en de gewenste draairichting van de cluster
END_REGION

REGION Network 11: +++ Berekeningen +++
   // Verscheidene berekeningen die nodig zijn voor de functionele werking of info voor weergave via de centrale en lokale bediening, zoals het  aantal bestuurbare ventilatoren, aantal ventilatoren aangestuurd in draairichting, actueel vermogen van de ventilatiecluster
END_REGION

REGION Network 12: +++ Bij- of afschakelen ventilator +++
   // Bijschakelen van de ventilator met het minst aantal draaiuren als aantal aangeschakelde ventilatoren lager dan het gewenst aantal. Afschakelen van de ventilator met meest aantal draaiuren als het aantal aangeschakelde ventilatoren hoger is dan het gewenst aantal.
END_REGION

REGION Network 13: +++ Automatische onderhoudstesten +++
   // Functionaliteit waarbij iedere ventilator een voor een aangestuurd wordt ter controle van de goede werking van iedere ventilator.
END_REGION

REGION Network 14: +++ Sturingen +++
   // Uitgeven van sturingen naar de ventilatoren.
END_REGION

REGION Network 15 (SCL): EINDE
   // Variabelen van intern scada rakvlak naar outputs copieren
   #VAR_CLUST.CAPA_OK := #VAR.CAPA_OK;
   #VAR_CLUST.NIV_AAN_BWA := #VAR.NIV_AAN_BWA;
   #VAR_CLUST.DIR := #VAR.DIR;
   #VAR_CLUST.BMO := #VAR.BMO;
   #VAR_CLUST.ONHD_STS := #VAR.ONHD_STS;
   #VAR_CLUST.PWR := #VAR.PWR;
END_REGION
END_FUNCTION_BLOCK

FUNCTION_BLOCK "TYPIC_C302_BF_LKM"   // FB68, FBD
TITLE = TYPIC_C302_BF_LKM: Luchtkwaliteitsmeting verkeerskoker
{ S7_Optimized_Access := 'TRUE' }
AUTHOR : OCOTECH
FAMILY : Typical
NAME : C302.801
// Logisch Object Besturing: C302.801
// 
// Het doel van de luchtkwaliteitsmeting is het meten van de zichtcondities in de verkeerskoker om op basis daarvan een indicatie te krijgen van de luchtkwaliteit in de verkeerskoker en rook in de verkeerskoker te detecteren.
// stored: MemoryReserve 10, SetENOAutomatically false
   VAR_INPUT
      STU_ALG_LCK_SIG { ExternalAccessible := 'False'; ExternalVisible := 'False'; ExternalWritable := 'False'} : USInt;   // Onderdruk alarmen
      CFG_SWA1 { ExternalAccessible := 'False'; ExternalVisible := 'False'; ExternalWritable := 'False'} : Real;   // Grenswaarde waarboven aangenomen wordt dat er lichte zichtbeperking is
      CFG_SWA2 { ExternalAccessible := 'False'; ExternalVisible := 'False'; ExternalWritable := 'False'} : Real;   // Grenswaarde waarboven aangenomen wordt dat er matige zichtbeperking is
      CFG_SWA3 { ExternalAccessible := 'False'; ExternalVisible := 'False'; ExternalWritable := 'False'} : Real;   // Grenswaarde waarboven aangenomen wordt dat er waarneembare zichtbeperking is
      CFG_SWA4 { ExternalAccessible := 'False'; ExternalVisible := 'False'; ExternalWritable := 'False'} : Real;   // Grenswaarde waarboven aangenomen wordt dat er ernstige zichtbeperking is
      CFG_HYS { ExternalAccessible := 'False'; ExternalVisible := 'False'; ExternalWritable := 'False'} : Real;   // Hysteresis om naar lagere aanduiding te gaan voor zichtkwaliteit
      CFG_MAX_NOK { ExternalAccessible := 'False'; ExternalVisible := 'False'; ExternalWritable := 'False'} : Int;   // Aantal opeenvolgende niet observeerbare luchtkwaliteitsmeters voor beschikbaarheidsstatus beperkt beschikbaar
   END_VAR
   VAR_OUTPUT
      VAR_ROOK { ExternalAccessible := 'False'; ExternalVisible := 'False'; ExternalWritable := 'False'} : USInt;   // Rookdetectie
      VAR_POS_ROOK { ExternalAccessible := 'False'; ExternalVisible := 'False'; ExternalWritable := 'False'} : Bool;   // Positie van de rookdetectie
      VAR_LKM_BWA { ExternalAccessible := 'False'; ExternalVisible := 'False'; ExternalWritable := 'False'} : Real;   // Meetwaarde luchtkwaliteit (maximumwaarde in koker)
   END_VAR
   VAR_IN_OUT
      VAR_LKM : Array[0..1] of Bool;   // Array met alle luchtkwaliteitsmeters, met alle variabelen van de luchtkwaliteitsmeter
   END_VAR
   VAR
      SIG { ExternalWritable := 'False'} : Struct   // Signaleringen
         AA01 : Bool;   // Openvolgende luchtkwaliteitsmeters niet observeerbaar
         AB01 : Bool;   // Luchtkwaliteitsmeting niet beschikbaar
         AB02 : Bool;   // Luchtkwaliteitsmeting beperkt beschikbaar
         AV01 : Bool;   // Rook gedetecteerd
         AV02 : Bool;   // Slecht zicht gedetecteerd
      END_STRUCT;
      VAR { ExternalWritable := 'False'} : Struct   // Variabelen
         BSC : USInt;   // Geeft de beschikbaarheid aan van de luchtkwaliteitsmeting aan
         VGV_SIG_VOP : Bool;   // TRUE = Signaleringen vrijgegeven voor verkeersoperator FALSE = Onderdrukt
         STS_BWA : USInt;   // Indicatie van de zichtbeperking (zichtconditie) in de tunnel
         POS { ExternalAccessible := 'False'; ExternalVisible := 'False'} : USInt;   // Positie in de tunnel van luchtkwaliteitsmeter die hoogste geldige k-waarde aangeeft
         "2oo3_BWA" { ExternalAccessible := 'False'; ExternalVisible := 'False'} : USInt;   // k-waarde als resultaat van 2oo3 filter
         "2oo3_POS" { ExternalAccessible := 'False'; ExternalVisible := 'False'} : USInt;   // Positie met hoogste k-waarde vanuit 2oo3 filter
         "2oo3_GEM" { ExternalAccessible := 'False'; ExternalVisible := 'False'} : USInt;   // Gemiddelde van de 3-metingen bij 2oo3 filter
         "2oo3_HULP1" { ExternalAccessible := 'False'; ExternalVisible := 'False'} : USInt;   // Gemiddelde van meting 2 en 3
         "2oo3_HULP2" { ExternalAccessible := 'False'; ExternalVisible := 'False'} : USInt;   // Gemiddelde van meting 1 en 3
         "2oo3_HULP3" { ExternalAccessible := 'False'; ExternalVisible := 'False'} : USInt;   // Gemiddelde van meting 1 en 2
         "2oo3_HULP4" { ExternalAccessible := 'False'; ExternalVisible := 'False'} : USInt;   // Procentuele afwijking HULP1 met GEM
         "2oo3_HULP5" { ExternalAccessible := 'False'; ExternalVisible := 'False'} : USInt;   // Procentuele afwijking HULP2 met GEM
         "2oo3_HULP6" { ExternalAccessible := 'False'; ExternalVisible := 'False'} : USInt;   // Procentuele afwijking HULP3 met GEM
         LKM_HULP { ExternalAccessible := 'False'; ExternalVisible := 'False'} : USInt;   // Hulpvariabele voor tussenresultaten
      END_STRUCT;
   END_VAR
BEGIN

REGION Network 1: START
END_REGION

REGION Network 2: +++ Bepalen meetwaarde luchtkwaliteitsmeting +++
   // Éen algemene meetwaarde voor de verkeerskoker bepalen op basis van de individuele metingen van alle luchtkwaliteitsmeters waarbij defecte luchtkwaliteitsmeters en afwijkende meetwaardes er uit gefilterd worden
END_REGION

REGION Network 3: +++ Indicatie zichtcondities +++
   // Zichtconditie in de verkeerskoker bepalen (Geen zichtbeperking / Lichte zichtbeperking / Matige zichtbeperking / Waarneembare zichtbeperking / Ernstige zichtbeperking).
END_REGION

REGION Network 4: +++ Rookdetectie +++
   // Aangeven van rookdetectie in de verkeerskoker en de lengtepositie in de verkeerskoker van de rookdetectie.
END_REGION

REGION Network 5: +++ Bepalen beschikbaarheidsstatus +++
   // Beschikbaarheidsstatus (beschikbaar / beperkt beschikbaar / niet beschikbaar) bepalen.
END_REGION

REGION Network 6 (SCL): Beschikbaarheidsstatus bepalen
   IF 
       //voorwaarden "Niet beschikbaar"
       TRUE
   THEN
       //Beschikbaarheidsstatus = Niet Beschikbaar
       #VAR.BSC:= "NietBeschikbaar";
   ELSIF
       //voorwaarden "Beperkt beschikbaar"
       TRUE
   THEN
       //Beschikbaarheidsstatus = Beperkt Beschikbaar
       #VAR.BSC:= "Beperkt";
   ELSE
       //Beschikbaarheidsstatus = Beschikbaar
       #VAR.BSC:= "Beschikbaar";
   END_IF;
END_REGION

REGION Network 7: +++ Signaleringen +++
   // Aanmaken signaleringen.
END_REGION

REGION Network 8: Signalering AB01 : Niet Beschikbaar
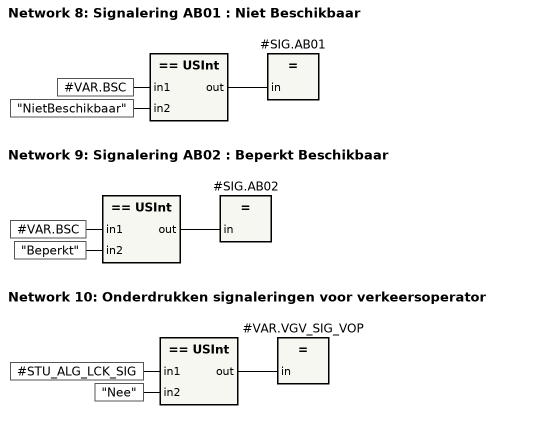
   #SIG.AB01 := #VAR.BSC = "NietBeschikbaar";
END_REGION

REGION Network 9: Signalering AB02 : Beperkt Beschikbaar
   #SIG.AB02 := #VAR.BSC = "Beperkt";
END_REGION

REGION Network 10: Onderdrukken signaleringen voor verkeersoperator
   // Via de variabele VGV_SIG_VOP wordt aan IRIS SCADA doorgegeven of signaleringen (bestemd voor de verkeersoperator) van de deze functie zichtbaar (of onderdrukt) moeten zijn.
   #VAR.VGV_SIG_VOP := #STU_ALG_LCK_SIG = "Nee";
END_REGION

REGION Network 11: EINDE
   // Variabelen van intern scada rakvlak naar outputs copieren
END_REGION
END_FUNCTION_BLOCK

FUNCTION_BLOCK "TYPIC_C302_IF_LKM"   // FB103, FBD
TITLE = TYPIC_C302_IF_LKM: Luchtkwaliteitsmeter
{ S7_Optimized_Access := 'TRUE' }
AUTHOR : OCOTECH
FAMILY : Typical
NAME : C302.701
// Logisch Object Besturing: C302.701
// 
// De interne functie luchtkwaliteitsmeting verzorgt de interne besturing en bewaking van een luchtkwaliteitsmeter.
// stored: MemoryReserve 10, SetENOAutomatically false
   VAR_INPUT
      EXT_AUT { ExternalAccessible := 'False'; ExternalVisible := 'False'; ExternalWritable := 'False'} : Bool;   // Externe (hoofd) beveiliging (1 = OK)
      EXT_HW { ExternalAccessible := 'False'; ExternalVisible := 'False'; ExternalWritable := 'False'} : Bool;   // Sturings hardware (PLC) bewaking (1 = OK)
      IN_AUT_C302 { ExternalAccessible := 'False'; ExternalVisible := 'False'; ExternalWritable := 'False'} : Bool;   // Beveiligingen: serie geschakelde terugmelding (1 = OK)
      IN_STS { ExternalAccessible := 'False'; ExternalVisible := 'False'; ExternalWritable := 'False'} : Bool;   // TRUE = Aan / FALSE = Uit
      IN_STO { ExternalAccessible := 'False'; ExternalVisible := 'False'; ExternalWritable := 'False'} : Bool;   // TRUE = OK / FALSE = Storing
      IN_MWA { ExternalAccessible := 'False'; ExternalVisible := 'False'; ExternalWritable := 'False'} : Word;   // Meetwaarde [m-1]
      CFG_MAX_SWA { ExternalAccessible := 'False'; ExternalVisible := 'False'; ExternalWritable := 'False'} : Real;   // Waarde doe toegekend wordt aan LKM_MWA als maximumwaarde voor de meeteenheid [m-1]
      CFG_MIN_SWA { ExternalAccessible := 'False'; ExternalVisible := 'False'; ExternalWritable := 'False'} : Real;   // Waarde doe toegekend wordt aan LKM_MWA als minimumwaarde voor de meeteenheid [m-1]
   END_VAR
   VAR_OUTPUT
      VAR_IF_LKM { ExternalAccessible := 'False'; ExternalVisible := 'False'; ExternalWritable := 'False'} : "C302_VAR_IF_LKM_TYPIC";   // Struct met alle variabelen naar bovenliggende functies
   END_VAR
   VAR
      STO { ExternalWritable := 'False'} : Struct   // Storingen
         A001 : Bool;   // Luchtkwaliteitsmeter niet aangeschakeld
         A002 : Bool;   // Draadbreuk analoge meting
         A003 : Bool;   // Meetbereik overschreden
         A004 : Bool;   // Luchtkwaliteitsmeter geeft storing
      END_STRUCT;
      VAR { ExternalWritable := 'False'} : Struct   // Variabelen
         LKM_MWA { ExternalAccessible := 'False'; ExternalVisible := 'False'} : Real;   // Meetwaarde [m-1]
         EXT_AUT { ExternalAccessible := 'False'; ExternalVisible := 'False'} : Bool;   // Externe (hoofd) beveiliging aangesproken
         EXT_HW { ExternalAccessible := 'False'; ExternalVisible := 'False'} : Bool;   // Sturings hardware (PLC) in storing
      END_STRUCT;
   END_VAR
BEGIN

REGION Network 1: START
END_REGION

REGION Network 2: +++ Verwerking analoge meting +++
   // Verwerking analoge meting naar een meetwaarde (k-waarde) en detectie storingen van de luchtkwaliteitsmeter.
END_REGION

REGION Network 3 (SCL): EINDE
   // Variabelen van intern scada rakvlak naar outputs copieren
   #VAR_IF_LKM.LKM_MWA := #VAR.LKM_MWA;
   #VAR_IF_LKM.EXT_AUT := #VAR.EXT_AUT;
   #VAR_IF_LKM.EXT_HW := #VAR.EXT_HW;
   #VAR_IF_LKM.STO := #STO;
END_REGION
END_FUNCTION_BLOCK

FUNCTION_BLOCK "TYPIC_C401_BF_RSS"   // FB105, FBD
TITLE = TYPIC_C401_BF_RSS: Rijstrooksignalisatie
{ S7_Optimized_Access := 'TRUE' }
AUTHOR : OCOTECH
FAMILY : Typical
NAME : C401.801
// Logisch Object Besturing: C401.801
// 
// De basisfunctie Rijstrooksignalisatie maakt een algemene status aan van de rijstrooksignalisatie voor een verkeerskoker.
// stored: MemoryReserve 10, SetENOAutomatically false
   VAR_INPUT
      CFG_MAX_NOK1 { ExternalAccessible := 'False'; ExternalVisible := 'False'; ExternalWritable := 'False'} : Int;   // Maximum aantal niet observeerbare RSS-borden ter voorkoming beschikbaarheidsstatus niet beschikbaar
      CFG_MAX_NOK2 { ExternalAccessible := 'False'; ExternalVisible := 'False'; ExternalWritable := 'False'} : Int;   // Maximum aantal opeenvolgende niet observeerbare RSS-borden per rijstrook ter voorkoming beschikbaarheidsstatus niet beschikbaar
      STU_ALG_LCK_SIG { ExternalAccessible := 'False'; ExternalVisible := 'False'; ExternalWritable := 'False'} : USInt;   // Onderdruk alarmen
   END_VAR
   VAR_IN_OUT
      VAR_RSS : Array[*] of "C401_VAR_RSS_TYPIC";   // Array van alle RSS-borden met een struct met alle variabelen van het RSS-bord
   END_VAR
   VAR
      SIG { ExternalWritable := 'False'} : Struct   // Signaleringen
         AB01 : Bool;   // Rijstrook signalisatie beperkt beschikbaar
         AB02 : Bool;   // Rijstrook signalisatie niet beschikbaar
      END_STRUCT;
      VAR { ExternalWritable := 'False'} : Struct   // Variabelen
         BSC : USInt;   // Geeft de beschikbaarheid aan van het rijstrooksignalisatie
         VGV_SIG_VOP : Bool;   // TRUE = Signaleringen vrijgegeven voor verkeersoperator FALSE = Onderdrukt
         AANT_NOK { ExternalAccessible := 'False'; ExternalVisible := 'False'} : USInt;   // Totaal aantal niet observeerbare RSS-borden
         MAX_NOK { ExternalAccessible := 'False'; ExternalVisible := 'False'} : USInt;   // Maximum gedetecteerd aantal opeenvolgende niet observeerbare RSS-borden per rijstrook
         HULP_NOK { ExternalAccessible := 'False'; ExternalVisible := 'False'} : USInt;   // Hulpvariabele voor maximum gedetecteerd aantal opeenvolgende niet observeerbare RSS-borden per rijstrook
         LUS_STO { ExternalAccessible := 'False'; ExternalVisible := 'False'} : USInt;   // OK = geen enkel luspaar geeft FOUT FOUT = een of meer lusparen geeft FOUT
      END_STRUCT;
   END_VAR
BEGIN

REGION Network 1: START
END_REGION

REGION Network 2: +++ Niet observeerbare RSS-borden en vaststelling luspaar storing +++
   // Deze functie omvat het tellen van het aantal RSS-borden dat niet observeerbaar is, tellen van het maximum aantal opeenvolgende RSS-borden dat niet observeerbaar is over een rijstrook en het vaststellen of er een luspaar een storing heeft.
END_REGION

REGION Network 3: +++ Bepalen beschikbaarheidsstatus +++
   // Beschikbaarheidsstatus (beschikbaar / beperkt beschikbaar / niet beschikbaar) bepalen.
END_REGION

REGION Network 4 (SCL): Beschikbaarheidsstatus bepalen
   IF 
       //voorwaarden "Niet beschikbaar"
       TRUE
   THEN
       //Beschikbaarheidsstatus = Niet Beschikbaar
       #VAR.BSC:= "NietBeschikbaar";
   ELSIF
       //voorwaarden "Beperkt beschikbaar"
       TRUE
   THEN
       //Beschikbaarheidsstatus = Beperkt Beschikbaar
       #VAR.BSC:= "Beperkt";
   ELSE
       //Beschikbaarheidsstatus = Beschikbaar
       #VAR.BSC:= "Beschikbaar";
   END_IF;
END_REGION

REGION Network 5: +++ Signaleringen +++
   // Aanmaken signaleringen.
END_REGION

REGION Network 6: Signalering AB01 : Niet Beschikbaar
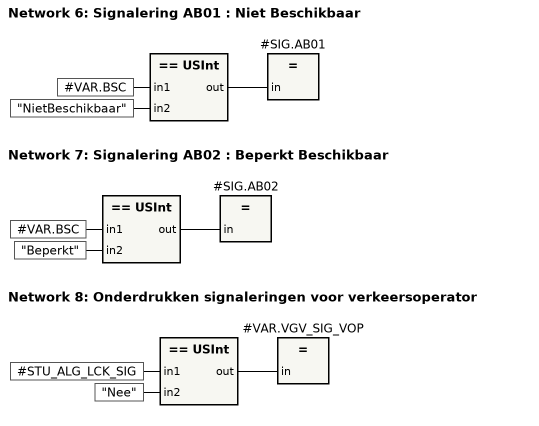
   #SIG.AB01 := #VAR.BSC = "NietBeschikbaar";
END_REGION

REGION Network 7: Signalering AB02 : Beperkt Beschikbaar
   #SIG.AB02 := #VAR.BSC = "Beperkt";
END_REGION

REGION Network 8: Onderdrukken signaleringen voor verkeersoperator
   // Via de variabele VGV_SIG_VOP wordt aan IRIS SCADA doorgegeven of signaleringen (bestemd voor de verkeersoperator) van de deze functie zichtbaar (of onderdrukt) moeten zijn.
   #VAR.VGV_SIG_VOP := #STU_ALG_LCK_SIG = "Nee";
END_REGION

REGION Network 9: EINDE
   // Variabelen van intern scada rakvlak naar outputs copieren
END_REGION
END_FUNCTION_BLOCK

